// TwinCAT 3 PLC project HOMS_XRT_PLC
// Title: lcls-plc-xrt-optics
// Company: SLAC
// ProjectVersion: 5.7.0
// ProgramVersion: 3.1.4022.7
// CompilerDefines: L
// libraries:
//   lcls-twincat-motion, * (SLAC)
//   lcls-twincat-optics, * (SLAC)
//   PMPS, * (SLAC - LCLS)
//   Tc2_ControllerToolbox, * (Beckhoff Automation GmbH)
//   Tc2_EtherCAT, * (Beckhoff Automation GmbH)
//   Tc2_MC2, * (Beckhoff Automation GmbH)
//   Tc2_SerialCom, * (Beckhoff Automation GmbH)
//   Tc2_Standard, * (Beckhoff Automation GmbH)
//   Tc2_System, * (Beckhoff Automation GmbH)
//   Tc2_Utilities, * (Beckhoff Automation GmbH)
//   Tc3_Module, * (Beckhoff Automation GmbH)
//   VisuDialogs, * (System)
//   LCLS General,2.8.2,SLAC
// project tree:
//   Common/DUTs/ ENUM_Coating_States.TcDUT, E_GantryControl.TcDUT, E_GantryMode.TcDUT, E_PiezoControl.TcDUT, E_PitchControl.TcDUT, HOMS_Gantry.TcDUT, HOMS_GantryAxis.TcDUT, HOMS_PitchMechanismOld.TcDUT, ST_AbstractAxis.TcDUT, ST_CoEIndSub.TcDUT, ST_DecoupledMotionPermits.TcDUT, ST_ElmoGDCBellCoEParams.TcDUT, ST_HOMSStepper.TcDUT, ST_PiezoAxisOld.TcDUT, ST_StepperStatus.TcDUT
//   Version/ Global_Version.TcGVL
//   Common/POUs/Helpers/ FB_Drive.TcPOU, FB_ElmoGDCBellCoE.TcPOU, FB_ElmoMCUploadDriveParams.TcPOU, FB_ElmoStoMonitor.TcPOU, FB_GantryDiffVirtualLimitSwitch.TcPOU, FB_InitDriveRefs.TcPOU, FB_LimitSwitchState.TcPOU, FB_PitchSoftLimits.TcPOU, FB_PI_E621_SerialDriverOld.TcPOU, FB_PI_E621_SerialTransaction.TcPOU, FB_PTP.TcPOU, FB_ReadFloatParameter.TcPOU, FB_ReadParameterInNC.TcPOU, FB_WriteParameterInNC.TcPOU, F_PiezoPosition.TcPOU, MC_SmoothMover.TcPOU, WithinRange.TcPOU
//   Common/POUs/HOMS_FBs/ FB_Gantry.TcPOU, FB_GantryDifferenceMonitor.TcPOU, FB_PiezoControl.TcPOU, FB_PitchControlOld.TcPOU, FB_ReduceGantryDiff.TcPOU
//   / GlobalTextList.TcGTLO, PiezoDriver.TcTTO, PlcTask.TcTTO, SerialIO.TcTTO, Visualization Manager.TcVMO (not stored)
//   GVLs/ GVL.TcGVL, GVL_COM_Buffers.TcGVL, GVL_Constants.TcGVL, GVL_MR1L3.TcGVL, GVL_MR1L4_Constants.TcGVL, GVL_MR1L4.TcGVL, GVL_MR1L3_Constants.TcGVL, GVL_MR2L3_Constants.TcGVL, GVL_MR2L3.TcGVL, GVL_PMPS.TcGVL, GVL_RTDS.TcGVL, GVL_SerialIO.TcGVL
//   POUs/ FB_Coating_States_noPMPS.TcPOU, FB_MirrorCoatingProtection.TcPOU, FB_Coating_States.TcPOU, Main.TcPOU, PRG_PMPS.TcPOU, PRG_CoatingProtection.TcPOU, PRG_States.TcPOU
//   POUs/Serial Comm/ PiezoSerial.TcPOU, P_Serial_Com.TcPOU
//   VISUs/ GantryControls.TcVIS, Visualization.TcVIS, PiezoControls.TcVIS
// real-time tasks:
//   TASK PlcTask: cycle T#10ms, priority 20, ADS port 350
//   TASK SerialIO: cycle T#2ms, priority 1, ADS port 351
//   TASK LoggerTask: cycle T#10ms, priority 2, ADS port 352
//   TASK PiezoDriver: cycle T#1ms, priority 3, ADS port 353
// motion (NC):
//   TASK NC-Task 1 SAF: cycle T#2ms, priority 4, ADS port 501
//   TASK NC-Task 1 SVB: cycle T#10ms, priority 8, ADS port 511
//   AXIS M1L3-Yup (id 1)
//     General: UnitName=um
//     Dynamic: Acceleration=200, Deceleration=200, DelayTime=0.008
//     Velo: Maximum=200
//     OtherSettings: AllowMotionCmdToSlave=true
//     encoder EncType=29
//       EncPara: ScaleFactorNumerator=0.001, Offset=-13611, MaxCount=#xffffffff
//         SoftEndMinControl: Enable=true, Range=-12130
//         SoftEndMaxControl: Enable=true, Range=12932
//         Inc: RefSoftSyncMask=#x0000ffff
//     drive DrvType=24
//       DrvPara: Inverse=true
//         Analog: VeloReferenz=488.28125, ScaleFactorActTorque=0.1
//         TimeComp: TaskDelayCycles=1
//     controller CtrType=2
//       CtrPara: PriorControlFactor=1
//         PosDiffControl: Range=100
//         PID: PosKp=50, PosExtKp=10, DeadBandPosition=0.3
//         Observer: BandWidth=20
//   AXIS M1L3-Ydwn (id 2)
//     General: UnitName=um
//     Dynamic: Acceleration=200, Deceleration=200, DelayTime=0.008
//     Velo: Maximum=200
//     OtherSettings: AllowMotionCmdToSlave=true
//     encoder EncType=29
//       EncPara: ScaleFactorNumerator=0.001, Offset=-13433.6, MaxCount=#xffffffff
//         SoftEndMinControl: Enable=true, Range=-12130
//         SoftEndMaxControl: Enable=true, Range=12932
//         Inc: RefSoftSyncMask=#x0000ffff
//     drive DrvType=24
//       DrvPara: Inverse=true
//         Analog: VeloReferenz=488.28125, ScaleFactorActTorque=0.1
//         TimeComp: TaskDelayCycles=1
//     controller CtrType=2
//       CtrPara: PriorControlFactor=1
//         PosDiffControl: Range=100
//         PID: PosKp=50, PosExtKp=10, DeadBandPosition=0.3
//         Observer: BandWidth=20
//   AXIS M1L3-Xup (id 3)
//     General: UnitName=um
//     Dynamic: Acceleration=2000, Deceleration=2000, DelayTime=0.008
//     Velo: Maximum=1000
//     OtherSettings: AllowMotionCmdToSlave=true
//     encoder EncType=29
//       EncPara: ScaleFactorNumerator=0.001, Offset=-25210.5, MaxCount=#xffffffff
//         SoftEndMinControl: Enable=true, Range=-6841
//         SoftEndMaxControl: Enable=true, Range=1452.7
//         Inc: RefSoftSyncMask=#x0000ffff
//     drive DrvType=24
//       Analog: VeloReferenz=1220.703125, ScaleFactorActTorque=0.1
//       TimeComp: TaskDelayCycles=1
//     controller CtrType=2
//       CtrPara: PriorControlFactor=1
//         PosDiffControl: Range=50
//         PID: PosKp=50, PosExtKp=50, DeadBandPosition=0.4
//         Observer: BandWidth=20
//   AXIS M1L3-Xdwn (id 4)
//     General: UnitName=um
//     Dynamic: Acceleration=2000, Deceleration=2000, DelayTime=0.008
//     Velo: Maximum=1000
//     OtherSettings: AllowMotionCmdToSlave=true
//     encoder EncType=29
//       EncPara: ScaleFactorNumerator=0.001, Offset=-24971.8, MaxCount=#xffffffff
//         SoftEndMinControl: Enable=true, Range=-6841.9
//         SoftEndMaxControl: Enable=true, Range=1452.7
//         Inc: RefSoftSyncMask=#x0000ffff
//     drive DrvType=24
//       DrvPara: Inverse=true
//         Analog: VeloReferenz=1220.703125, ScaleFactorActTorque=0.1
//         TimeComp: TaskDelayCycles=1
//     controller CtrType=2
//       CtrPara: PriorControlFactor=1
//         PosDiffControl: Range=50
//         PID: PosKp=50, PosExtKp=50, DeadBandPosition=0.4
//         Observer: BandWidth=20
//   AXIS M1L3-Pitch (id 5)
//     General: UnitName=urad
//     Dynamic: Acceleration=390, Deceleration=390, DelayTime=0.008
//     Velo: Maximum=150
//     OtherSettings: AllowMotionCmdToSlave=true
//     encoder EncType=29
//       EncPara: ScaleFactorNumerator=0.001949317739, Offset=-21644.29, MaxCount=#xffffffff
//         FilterTime: TPos=0.2
//         SoftEndMinControl: Enable=true, Range=-193
//         SoftEndMaxControl: Enable=true, Range=220
//         Inc: RefSoftSyncMask=#x0000ffff
//     drive DrvType=24
//       Analog: VeloReferenz=371.8028524, ScaleFactorActTorque=0.1
//       TimeComp: TaskDelayCycles=1
//     controller CtrType=2
//       CtrPara: PriorControlFactor=1
//         PosDiffControl: Range=30
//         PID: PosKp=2, PosExtKp=1, DeadBandPosition=0.01
//         Observer: BandWidth=20
//   AXIS M1L3-Bender (id 6)
//     General: UnitName=um
//     Dynamic: Acceleration=150, Deceleration=150, DelayTime=0.008
//     Velo: Maximum=150
//     OtherSettings: AllowMotionCmdToSlave=true
//     encoder EncType=29
//       EncPara: ScaleFactorNumerator=0.001, MaxCount=#xffffffff
//         SoftEndMinControl: Enable=true, Range=18000
//         SoftEndMaxControl: Enable=true, Range=27800
//         Inc: RefSoftSyncMask=#x0000ffff
//     drive DrvType=24
//       DrvPara: Inverse=true
//         Analog: VeloReferenz=150, ScaleFactorActTorque=0.1
//         TimeComp: TaskDelayCycles=1
//     controller CtrType=2
//       CtrPara: PriorControlFactor=1
//         PID: PosKp=10, PosExtKp=0.001, PosExtVelo=0.9, DeadBandPosition=0.1
//         Observer: BandWidth=20
//   AXIS M2L3-Yup (id 13)
//     General: UnitName=um
//     Dynamic: Acceleration=200, Deceleration=200, DelayTime=0.008
//     Velo: Maximum=200
//     OtherSettings: AllowMotionCmdToSlave=true
//     encoder EncType=29
//       EncPara: ScaleFactorNumerator=0.001, Offset=-14279, MaxCount=#xffffffff
//         SoftEndMinControl: Enable=true, Range=-11750
//         SoftEndMaxControl: Enable=true, Range=12530
//         Inc: RefSoftSyncMask=#x0000ffff
//     drive DrvType=24
//       DrvPara: Inverse=true
//         Analog: VeloReferenz=488.28125, ScaleFactorActTorque=0.1
//         TimeComp: TaskDelayCycles=1
//     controller CtrType=2
//       CtrPara: PriorControlFactor=1
//         PosDiffControl: Range=100
//         PID: PosKp=50, PosExtKp=10, DeadBandPosition=0.3
//         Observer: BandWidth=20
//   AXIS M2L3-Ydwn (id 14)
//     General: UnitName=um
//     Dynamic: Acceleration=200, Deceleration=200, DelayTime=0.008
//     Velo: Maximum=200
//     OtherSettings: AllowMotionCmdToSlave=true
//     encoder EncType=29
//       EncPara: ScaleFactorNumerator=0.001, Offset=-16314.1, MaxCount=#xffffffff
//         SoftEndMinControl: Enable=true, Range=-11750
//         SoftEndMaxControl: Enable=true, Range=12531.5
//         Inc: RefSoftSyncMask=#x0000ffff
//     drive DrvType=24
//       DrvPara: Inverse=true
//         Analog: VeloReferenz=488.28125, ScaleFactorActTorque=0.1
//         TimeComp: TaskDelayCycles=1
//     controller CtrType=2
//       CtrPara: PriorControlFactor=1
//         PosDiffControl: Range=100
//         PID: PosKp=50, PosExtKp=10, DeadBandPosition=0.3
//         Observer: BandWidth=20
//   AXIS M2L3-Xup (id 15)
//     General: UnitName=um
//     Dynamic: Acceleration=2000, Deceleration=2000, DelayTime=0.008
//     Velo: Maximum=1000
//     OtherSettings: AllowMotionCmdToSlave=true
//     encoder EncType=29
//       EncPara: ScaleFactorNumerator=0.001, Offset=-25135.5, MaxCount=#xffffffff
//         SoftEndMinControl: Enable=true, Range=-850
//         SoftEndMaxControl: Enable=true, Range=867.4
//         Inc: RefSoftSyncMask=#x0000ffff
//     drive DrvType=24
//       Analog: VeloReferenz=1220.703125, ScaleFactorActTorque=0.1
//       TimeComp: TaskDelayCycles=1
//     controller CtrType=2
//       CtrPara: PriorControlFactor=1
//         PosDiffControl: Range=50
//         PID: PosKp=50, PosExtKp=50, DeadBandPosition=0.4
//         Observer: BandWidth=20
//   AXIS M2L3-Xdwn (id 16)
//     General: UnitName=um
//     Dynamic: Acceleration=2000, Deceleration=2000, DelayTime=0.008
//     Velo: Maximum=1000
//     OtherSettings: AllowMotionCmdToSlave=true
//     encoder EncType=29
//       EncPara: ScaleFactorNumerator=0.001, Offset=-24091, MaxCount=#xffffffff
//         SoftEndMinControl: Enable=true, Range=-865
//         SoftEndMaxControl: Enable=true, Range=862.6
//         Inc: RefSoftSyncMask=#x0000ffff
//     drive DrvType=24
//       DrvPara: Inverse=true
//         Analog: VeloReferenz=1220.703125, ScaleFactorActTorque=0.1
//         TimeComp: TaskDelayCycles=1
//     controller CtrType=2
//       CtrPara: PriorControlFactor=1
//         PosDiffControl: Range=50
//         PID: PosKp=50, PosExtKp=50, DeadBandPosition=0.4
//         Observer: BandWidth=20
//   AXIS M2L3-Pitch (id 17)
//     General: UnitName=urad
//     Dynamic: Acceleration=390, Deceleration=390, DelayTime=0.008
//     Velo: Maximum=150
//     OtherSettings: AllowMotionCmdToSlave=true
//     encoder EncType=29
//       EncPara: ScaleFactorNumerator=0.001949317739, Offset=-17539, MaxCount=#xffffffff
//         FilterTime: TPos=0.2
//         SoftEndMinControl: Enable=true, Range=-212
//         SoftEndMaxControl: Enable=true, Range=246
//         Inc: RefSoftSyncMask=#x0000ffff
//     drive DrvType=24
//       Analog: VeloReferenz=371.8028524, ScaleFactorActTorque=0.1
//       TimeComp: TaskDelayCycles=1
//     controller CtrType=2
//       CtrPara: PriorControlFactor=1
//         PosDiffControl: Range=15
//         PID: PosKp=2, PosExtKp=1, DeadBandPosition=0.01
//         Observer: BandWidth=20
//   AXIS M2L3-Bender (id 18)
//     General: UnitName=um
//     Dynamic: Acceleration=150, Deceleration=150, DelayTime=0.008
//     Velo: Maximum=150
//     OtherSettings: AllowMotionCmdToSlave=true
//     encoder EncType=29
//       EncPara: ScaleFactorNumerator=0.001, MaxCount=#xffffffff
//         SoftEndMinControl: Enable=true, Range=20000
//         SoftEndMaxControl: Enable=true, Range=32000
//         Inc: RefSoftSyncMask=#x0000ffff
//     drive DrvType=24
//       DrvPara: Inverse=true
//         Analog: VeloReferenz=195.3125, ScaleFactorActTorque=0.1
//         TimeComp: TaskDelayCycles=1
//     controller CtrType=2
//       CtrPara: PriorControlFactor=1
//         PID: PosKp=10, PosExtKp=0.001, PosExtVelo=0.9, DeadBandPosition=0.1
//         Observer: BandWidth=20
//   AXIS M1L4-Yup (id 7)
//     General: UnitName=um
//     Dynamic: Acceleration=200, Deceleration=200, DelayTime=0.008
//     Velo: Maximum=200
//     OtherSettings: AllowMotionCmdToSlave=true
//     encoder EncType=29
//       EncPara: ScaleFactorNumerator=0.001, Offset=-13496.029, MaxCount=#xffffffff
//         SoftEndMinControl: Enable=true, Range=-11000
//         SoftEndMaxControl: Enable=true, Range=12000
//         Inc: RefSoftSyncMask=#x0000ffff
//     drive DrvType=24
//       DrvPara: Inverse=true
//         Analog: VeloReferenz=488.28125, ScaleFactorActTorque=0.1
//         TimeComp: TaskDelayCycles=1
//     controller CtrType=2
//       CtrPara: PriorControlFactor=1
//         PosDiffControl: Range=100
//         PID: PosKp=50, PosExtKp=10, DeadBandPosition=0.3
//         Observer: BandWidth=20
//   AXIS M1L4-Ydwn (id 8)
//     General: UnitName=um
//     Dynamic: Acceleration=200, Deceleration=200, DelayTime=0.008
//     Velo: Maximum=200
//     OtherSettings: AllowMotionCmdToSlave=true
//     encoder EncType=29
//       EncPara: ScaleFactorNumerator=0.001, Offset=-14872.55, MaxCount=#xffffffff
//         SoftEndMinControl: Enable=true, Range=-11000
//         SoftEndMaxControl: Enable=true, Range=12075
//         Inc: RefSoftSyncMask=#x0000ffff
//     drive DrvType=24
//       DrvPara: Inverse=true
//         Analog: VeloReferenz=488.28125, ScaleFactorActTorque=0.1
//         TimeComp: TaskDelayCycles=1
//     controller CtrType=2
//       CtrPara: PriorControlFactor=1
//         PosDiffControl: Range=100
//         PID: PosKp=50, PosExtKp=10, DeadBandPosition=0.3
//         Observer: BandWidth=20
//   AXIS M1L4-Xup (id 9)
//     General: UnitName=um
//     Dynamic: Acceleration=2000, Deceleration=2000, DelayTime=0.008
//     Velo: Maximum=1000
//     OtherSettings: AllowMotionCmdToSlave=true
//     encoder EncType=29
//       EncPara: ScaleFactorNumerator=0.001, Offset=-25490.849, MaxCount=#xffffffff
//         SoftEndMinControl: Enable=true, Range=-2000
//         SoftEndMaxControl: Enable=true, Range=18750
//         Inc: RefSoftSyncMask=#x0000ffff
//     drive DrvType=24
//       Analog: VeloReferenz=1220.703125, ScaleFactorActTorque=0.1
//       TimeComp: TaskDelayCycles=1
//     controller CtrType=2
//       CtrPara: PriorControlFactor=1
//         PosDiffControl: Range=50
//         PID: PosKp=50, PosExtKp=50, DeadBandPosition=0.4
//         Observer: BandWidth=20
//   AXIS M1L4-Xdwn (id 10)
//     General: UnitName=um
//     Dynamic: Acceleration=2000, Deceleration=2000, DelayTime=0.008
//     Velo: Maximum=1000
//     OtherSettings: AllowMotionCmdToSlave=true
//     encoder EncType=29
//       EncPara: ScaleFactorNumerator=0.001, Offset=-26628.83, MaxCount=#xffffffff
//         SoftEndMinControl: Enable=true, Range=-2050
//         SoftEndMaxControl: Enable=true, Range=18750
//         Inc: RefSoftSyncMask=#x0000ffff
//     drive DrvType=24
//       DrvPara: Inverse=true
//         Analog: VeloReferenz=1220.703125, ScaleFactorActTorque=0.1
//         TimeComp: TaskDelayCycles=1
//     controller CtrType=2
//       CtrPara: PriorControlFactor=1
//         PosDiffControl: Range=50
//         PID: PosKp=50, PosExtKp=50, DeadBandPosition=0.4
//         Observer: BandWidth=20
//   AXIS M1L4-Pitch (id 11)
//     General: UnitName=urad
//     Dynamic: Acceleration=390, Deceleration=390, DelayTime=0.008
//     Velo: Maximum=150
//     OtherSettings: AllowMotionCmdToSlave=true
//     encoder EncType=29
//       EncPara: ScaleFactorNumerator=0.001949317739, Offset=-19152.5, MaxCount=#xffffffff
//         FilterTime: TPos=0.2
//         SoftEndMinControl: Enable=true, Range=-900
//         SoftEndMaxControl: Enable=true, Range=900
//         Inc: RefSoftSyncMask=#x0000ffff
//     drive DrvType=24
//       Analog: VeloReferenz=371.8028524, ScaleFactorActTorque=0.1
//       TimeComp: TaskDelayCycles=1
//     controller CtrType=2
//       CtrPara: PriorControlFactor=1
//         PosDiffControl: Range=30
//         PID: PosKp=2, PosExtKp=1, DeadBandPosition=0.01
//         Observer: BandWidth=20
//   AXIS M1L4-Bender (id 12)
//     General: UnitName=um
//     Dynamic: AccelerationMaximum=50, DecelerationMaximum=50, Acceleration=50, Deceleration=50, DelayTime=0.008
//     Velo: Maximum=150
//     OtherSettings: AllowMotionCmdToSlave=true
//     encoder EncType=29
//       EncPara: ScaleFactorNumerator=0.001, Offset=-4295012.99, MaxCount=#xffffffff
//         SoftEndMinControl: Enable=true, Range=-26500
//         SoftEndMaxControl: Enable=true, Range=-16500
//     drive DrvType=24
//       DrvPara: Inverse=true
//         Analog: VeloReferenz=195.3125, ScaleFactorActTorque=0.1
//         TimeComp: TaskDelayCycles=1
//     controller CtrType=2
//       CtrPara: PriorControlFactor=1
//         PosDiffControl: Range=100
//         PID: PosKp=10, PosExtKp=0.001, PosExtVelo=0.9, DeadBandPosition=0.1
//         Observer: BandWidth=20
// I/O:
//   DEVICE HOMS, AmsNetId 172.21.88.136.2.1
//     Term 1 (EK1200) [EK1200-5000 EtherCAT Power supply (2A E-Bus)]
//       Term 24 (EL9187) [EL9187 Potential Connection, 8 x Ground]
//       Term 13 (EL2008) [EL2008 8Ch. Dig. Output 24V, 0.5A]
//       Term 14 (EK1122) [EK1122 2 port EtherCAT junction]
//         EK1100_M1L3 [EK1100 EtherCAT Coupler (2A E-Bus)]
//           EL7041-1000_M1L3_Xup [EL7041-1000 1Ch. Stepper motor output stage (50V, 5A, standard)]
//           EL7041-1000_M1L3_Xdwn [EL7041-1000 1Ch. Stepper motor output stage (50V, 5A, standard)]
//           EL7041-1000_M1L3_Yup [EL7041-1000 1Ch. Stepper motor output stage (50V, 5A, standard)]
//           EL7041-1000_M1L3_Ydwn [EL7041-1000 1Ch. Stepper motor output stage (50V, 5A, standard)]
//           EL7041-1000_M1L3_PitchCoarse [EL7041-1000 1Ch. Stepper motor output stage (50V, 5A, standard)]
//           EL7041-1000_M1L3_Bender
//           EL6001_M1L3_PitchFine [EL6001 Interface (RS232)]
//           EL5042_M1L3_Xupdwn
//           EL5042_M1L3_Yupdwn
//           EL5042_M1L3_PitchBender
//           EL1004_M1L3_STO
//           EL9505_M1L3_BenderLims
//           MR1L3-EL3202-0010-E13
//           MR1L3-EL3202-0010-E14
//           Term 42 (EL9011)
//         EK1100_M1L4 [EK1100 EtherCAT Coupler (2A E-Bus)]
//           EL7041-1000_M1L4_Xup [EL7041-1000 1Ch. Stepper motor output stage (50V, 5A, standard)]
//           EL7041-1000_M1L4_Xdwn [EL7041-1000 1Ch. Stepper motor output stage (50V, 5A, standard)]
//           EL7041-1000_M1L4_Yup [EL7041-1000 1Ch. Stepper motor output stage (50V, 5A, standard)]
//           EL7041-1000_M1L4_Ydwn [EL7041-1000 1Ch. Stepper motor output stage (50V, 5A, standard)]
//           EL7041-1000_M1L4_PitchCoarse [EL7041-1000 1Ch. Stepper motor output stage (50V, 5A, standard)]
//           EL7041-1000_M1L4_Bender
//           EL6001_M1L4_PitchFine [EL6001 Interface (RS232)]
//           EL5042_M1L4_Xupdwn
//           EL5042_M1L4_Yupdwn
//           EL5042_M1L4_PitchBender
//           EL1004_M1L4_STO
//           EL9505_M1L4_BenderLims
//           MR1L4-EL3202-0010-E13
//           MR1L4-EL3202-0010-E14
//           Term 29 (EL9011)
//       Term 2 (EK1122) [EK1122 2 port EtherCAT junction]
//         EK1100_M2L3
//       Term 34 (EK1521-0010)
// variable links:
//   (this object) <-> HOMS/Term 1 (EK1200)/Term 14 (EK1122)/EK1100_M1L3/EL5042_M1L3_Yupdwn
//     Enc/Inputs/In/nComState @bit 1 <-> WcState/InputToggle
//     Enc/Inputs/In/nComState <-> WcState/WcState
//     Enc/Inputs/In/nDataIn1 <-> FB Inputs Channel 1/Position
//     Enc/Inputs/In/nDataIn1 <-> FB Inputs Channel 2/Position
//     Enc/Inputs/In/nState1 @bit 12 <-> FB Inputs Channel 1/Status/Diag
//     Enc/Inputs/In/nState1 @bit 12 <-> FB Inputs Channel 2/Status/Diag
//     Enc/Inputs/In/nState1 @bit 1 <-> FB Inputs Channel 1/Status/Error
//     Enc/Inputs/In/nState1 @bit 1 <-> FB Inputs Channel 2/Status/Error
//     Enc/Inputs/In/nState1 @bit 14 <-> FB Inputs Channel 1/Status/Input cycle counter
//     Enc/Inputs/In/nState1 @bit 14 <-> FB Inputs Channel 2/Status/Input cycle counter
//     Enc/Inputs/In/nState1 @bit 2 <-> FB Inputs Channel 1/Status/Ready
//     Enc/Inputs/In/nState1 @bit 2 <-> FB Inputs Channel 2/Status/Ready
//     Enc/Inputs/In/nState1 @bit 13 <-> FB Inputs Channel 1/Status/TxPDO State
//     Enc/Inputs/In/nState1 @bit 13 <-> FB Inputs Channel 2/Status/TxPDO State
//     Enc/Inputs/In/nState1 <-> FB Inputs Channel 1/Status/Warning
//     Enc/Inputs/In/nState1 <-> FB Inputs Channel 2/Status/Warning
//   (this object) <-> HOMS/Term 1 (EK1200)/Term 14 (EK1122)/EK1100_M1L3/EL7041-1000_M1L3_Yup
//     Drive/Inputs/In/nState1 @bit 3 <-> STM Status/Status/Error
//     Drive/Inputs/In/nState1 @bit 5 <-> STM Status/Status/Moving negative
//     Drive/Inputs/In/nState1 @bit 4 <-> STM Status/Status/Moving positive
//     Drive/Inputs/In/nState1 @bit 1 <-> STM Status/Status/Ready
//     Drive/Inputs/In/nState1 <-> STM Status/Status/Ready to enable
//     Drive/Inputs/In/nState1 @bit 6 <-> STM Status/Status/Torque reduced
//     Drive/Inputs/In/nState1 @bit 2 <-> STM Status/Status/Warning
//     Drive/Inputs/In/nState2 @bit 3 <-> STM Status/Status/Digital input 1
//     Drive/Inputs/In/nState2 @bit 4 <-> STM Status/Status/Digital input 2
//     Drive/Inputs/In/nState2 @bit 5 <-> STM Status/Status/Sync error
//     Drive/Inputs/In/nState2 @bit 7 <-> STM Status/Status/TxPDO Toggle
//     Drive/Inputs/In/nState4 @bit 1 <-> WcState/InputToggle
//     Drive/Inputs/In/nState4 <-> WcState/WcState
//     Drive/Outputs/Out/nCtrl1 <-> STM Control/Control/Enable
//     Drive/Outputs/Out/nCtrl1 @bit 2 <-> STM Control/Control/Reduce torque
//     Drive/Outputs/Out/nCtrl1 @bit 1 <-> STM Control/Control/Reset
//     Drive/Outputs/Out/nDataOut2[0] <-> STM Velocity/Velocity
//   (this object) <-> HOMS/Term 1 (EK1200)/Term 14 (EK1122)/EK1100_M1L3/EL7041-1000_M1L3_Ydwn
//     Drive/Inputs/In/nState1 @bit 3 <-> STM Status/Status/Error
//     Drive/Inputs/In/nState1 @bit 5 <-> STM Status/Status/Moving negative
//     Drive/Inputs/In/nState1 @bit 4 <-> STM Status/Status/Moving positive
//     Drive/Inputs/In/nState1 @bit 1 <-> STM Status/Status/Ready
//     Drive/Inputs/In/nState1 <-> STM Status/Status/Ready to enable
//     Drive/Inputs/In/nState1 @bit 6 <-> STM Status/Status/Torque reduced
//     Drive/Inputs/In/nState1 @bit 2 <-> STM Status/Status/Warning
//     Drive/Inputs/In/nState2 @bit 3 <-> STM Status/Status/Digital input 1
//     Drive/Inputs/In/nState2 @bit 4 <-> STM Status/Status/Digital input 2
//     Drive/Inputs/In/nState2 @bit 5 <-> STM Status/Status/Sync error
//     Drive/Inputs/In/nState2 @bit 7 <-> STM Status/Status/TxPDO Toggle
//     Drive/Inputs/In/nState4 @bit 1 <-> WcState/InputToggle
//     Drive/Inputs/In/nState4 <-> WcState/WcState
//     Drive/Outputs/Out/nCtrl1 <-> STM Control/Control/Enable
//     Drive/Outputs/Out/nCtrl1 @bit 2 <-> STM Control/Control/Reduce torque
//     Drive/Outputs/Out/nCtrl1 @bit 1 <-> STM Control/Control/Reset
//     Drive/Outputs/Out/nDataOut2[0] <-> STM Velocity/Velocity
//   (this object) <-> HOMS/Term 1 (EK1200)/Term 14 (EK1122)/EK1100_M1L3/EL5042_M1L3_Xupdwn
//     Enc/Inputs/In/nComState @bit 1 <-> WcState/InputToggle
//     Enc/Inputs/In/nComState <-> WcState/WcState
//     Enc/Inputs/In/nDataIn1 <-> FB Inputs Channel 1/Position
//     Enc/Inputs/In/nDataIn1 <-> FB Inputs Channel 2/Position
//     Enc/Inputs/In/nState1 @bit 12 <-> FB Inputs Channel 1/Status/Diag
//     Enc/Inputs/In/nState1 @bit 12 <-> FB Inputs Channel 2/Status/Diag
//     Enc/Inputs/In/nState1 @bit 1 <-> FB Inputs Channel 1/Status/Error
//     Enc/Inputs/In/nState1 @bit 1 <-> FB Inputs Channel 2/Status/Error
//     Enc/Inputs/In/nState1 @bit 14 <-> FB Inputs Channel 1/Status/Input cycle counter
//     Enc/Inputs/In/nState1 @bit 14 <-> FB Inputs Channel 2/Status/Input cycle counter
//     Enc/Inputs/In/nState1 @bit 2 <-> FB Inputs Channel 1/Status/Ready
//     Enc/Inputs/In/nState1 @bit 2 <-> FB Inputs Channel 2/Status/Ready
//     Enc/Inputs/In/nState1 @bit 13 <-> FB Inputs Channel 1/Status/TxPDO State
//     Enc/Inputs/In/nState1 @bit 13 <-> FB Inputs Channel 2/Status/TxPDO State
//     Enc/Inputs/In/nState1 <-> FB Inputs Channel 1/Status/Warning
//     Enc/Inputs/In/nState1 <-> FB Inputs Channel 2/Status/Warning
//   (this object) <-> HOMS/Term 1 (EK1200)/Term 14 (EK1122)/EK1100_M1L3/EL7041-1000_M1L3_Xup
//     Drive/Inputs/In/nState1 @bit 3 <-> STM Status/Status/Error
//     Drive/Inputs/In/nState1 @bit 5 <-> STM Status/Status/Moving negative
//     Drive/Inputs/In/nState1 @bit 4 <-> STM Status/Status/Moving positive
//     Drive/Inputs/In/nState1 @bit 1 <-> STM Status/Status/Ready
//     Drive/Inputs/In/nState1 <-> STM Status/Status/Ready to enable
//     Drive/Inputs/In/nState1 @bit 6 <-> STM Status/Status/Torque reduced
//     Drive/Inputs/In/nState1 @bit 2 <-> STM Status/Status/Warning
//     Drive/Inputs/In/nState2 @bit 3 <-> STM Status/Status/Digital input 1
//     Drive/Inputs/In/nState2 @bit 4 <-> STM Status/Status/Digital input 2
//     Drive/Inputs/In/nState2 @bit 5 <-> STM Status/Status/Sync error
//     Drive/Inputs/In/nState2 @bit 7 <-> STM Status/Status/TxPDO Toggle
//     Drive/Inputs/In/nState4 @bit 1 <-> WcState/InputToggle
//     Drive/Inputs/In/nState4 <-> WcState/WcState
//     Drive/Outputs/Out/nCtrl1 <-> STM Control/Control/Enable
//     Drive/Outputs/Out/nCtrl1 @bit 2 <-> STM Control/Control/Reduce torque
//     Drive/Outputs/Out/nCtrl1 @bit 1 <-> STM Control/Control/Reset
//     Drive/Outputs/Out/nDataOut2[0] <-> STM Velocity/Velocity
//   (this object) <-> HOMS/Term 1 (EK1200)/Term 14 (EK1122)/EK1100_M1L3/EL7041-1000_M1L3_Xdwn
//     Drive/Inputs/In/nState1 @bit 3 <-> STM Status/Status/Error
//     Drive/Inputs/In/nState1 @bit 5 <-> STM Status/Status/Moving negative
//     Drive/Inputs/In/nState1 @bit 4 <-> STM Status/Status/Moving positive
//     Drive/Inputs/In/nState1 @bit 1 <-> STM Status/Status/Ready
//     Drive/Inputs/In/nState1 <-> STM Status/Status/Ready to enable
//     Drive/Inputs/In/nState1 @bit 6 <-> STM Status/Status/Torque reduced
//     Drive/Inputs/In/nState1 @bit 2 <-> STM Status/Status/Warning
//     Drive/Inputs/In/nState2 @bit 3 <-> STM Status/Status/Digital input 1
//     Drive/Inputs/In/nState2 @bit 4 <-> STM Status/Status/Digital input 2
//     Drive/Inputs/In/nState2 @bit 5 <-> STM Status/Status/Sync error
//     Drive/Inputs/In/nState2 @bit 7 <-> STM Status/Status/TxPDO Toggle
//     Drive/Inputs/In/nState4 @bit 1 <-> WcState/InputToggle
//     Drive/Inputs/In/nState4 <-> WcState/WcState
//     Drive/Outputs/Out/nCtrl1 <-> STM Control/Control/Enable
//     Drive/Outputs/Out/nCtrl1 @bit 2 <-> STM Control/Control/Reduce torque
//     Drive/Outputs/Out/nCtrl1 @bit 1 <-> STM Control/Control/Reset
//     Drive/Outputs/Out/nDataOut2[0] <-> STM Velocity/Velocity
//   (this object) <-> HOMS/Term 1 (EK1200)/Term 14 (EK1122)/EK1100_M1L3/EL5042_M1L3_PitchBender
//     Enc/Inputs/In/nComState @bit 1 <-> WcState/InputToggle
//     Enc/Inputs/In/nComState <-> WcState/WcState
//     Enc/Inputs/In/nDataIn1 <-> FB Inputs Channel 1/Position
//     Enc/Inputs/In/nDataIn1 <-> FB Inputs Channel 2/Position
//     Enc/Inputs/In/nState1 @bit 12 <-> FB Inputs Channel 1/Status/Diag
//     Enc/Inputs/In/nState1 @bit 12 <-> FB Inputs Channel 2/Status/Diag
//     Enc/Inputs/In/nState1 @bit 1 <-> FB Inputs Channel 1/Status/Error
//     Enc/Inputs/In/nState1 @bit 1 <-> FB Inputs Channel 2/Status/Error
//     Enc/Inputs/In/nState1 @bit 14 <-> FB Inputs Channel 1/Status/Input cycle counter
//     Enc/Inputs/In/nState1 @bit 14 <-> FB Inputs Channel 2/Status/Input cycle counter
//     Enc/Inputs/In/nState1 @bit 2 <-> FB Inputs Channel 1/Status/Ready
//     Enc/Inputs/In/nState1 @bit 2 <-> FB Inputs Channel 2/Status/Ready
//     Enc/Inputs/In/nState1 @bit 13 <-> FB Inputs Channel 1/Status/TxPDO State
//     Enc/Inputs/In/nState1 @bit 13 <-> FB Inputs Channel 2/Status/TxPDO State
//     Enc/Inputs/In/nState1 <-> FB Inputs Channel 1/Status/Warning
//     Enc/Inputs/In/nState1 <-> FB Inputs Channel 2/Status/Warning
//   (this object) <-> HOMS/Term 1 (EK1200)/Term 14 (EK1122)/EK1100_M1L3/EL7041-1000_M1L3_PitchCoarse
//     Drive/Inputs/In/nState1 @bit 3 <-> STM Status/Status/Error
//     Drive/Inputs/In/nState1 @bit 5 <-> STM Status/Status/Moving negative
//     Drive/Inputs/In/nState1 @bit 4 <-> STM Status/Status/Moving positive
//     Drive/Inputs/In/nState1 @bit 1 <-> STM Status/Status/Ready
//     Drive/Inputs/In/nState1 <-> STM Status/Status/Ready to enable
//     Drive/Inputs/In/nState1 @bit 6 <-> STM Status/Status/Torque reduced
//     Drive/Inputs/In/nState1 @bit 2 <-> STM Status/Status/Warning
//     Drive/Inputs/In/nState2 @bit 3 <-> STM Status/Status/Digital input 1
//     Drive/Inputs/In/nState2 @bit 4 <-> STM Status/Status/Digital input 2
//     Drive/Inputs/In/nState2 @bit 5 <-> STM Status/Status/Sync error
//     Drive/Inputs/In/nState2 @bit 7 <-> STM Status/Status/TxPDO Toggle
//     Drive/Inputs/In/nState4 @bit 1 <-> WcState/InputToggle
//     Drive/Inputs/In/nState4 <-> WcState/WcState
//     Drive/Outputs/Out/nCtrl1 <-> STM Control/Control/Enable
//     Drive/Outputs/Out/nCtrl1 @bit 2 <-> STM Control/Control/Reduce torque
//     Drive/Outputs/Out/nCtrl1 @bit 1 <-> STM Control/Control/Reset
//     Drive/Outputs/Out/nDataOut2[0] <-> STM Velocity/Velocity
//   (this object) <-> HOMS/Term 1 (EK1200)/Term 14 (EK1122)/EK1100_M1L3/EL7041-1000_M1L3_Bender
//     Drive/Inputs/In/nState1 @bit 3 <-> STM Status/Status/Error
//     Drive/Inputs/In/nState1 @bit 5 <-> STM Status/Status/Moving negative
//     Drive/Inputs/In/nState1 @bit 4 <-> STM Status/Status/Moving positive
//     Drive/Inputs/In/nState1 @bit 1 <-> STM Status/Status/Ready
//     Drive/Inputs/In/nState1 <-> STM Status/Status/Ready to enable
//     Drive/Inputs/In/nState1 @bit 6 <-> STM Status/Status/Torque reduced
//     Drive/Inputs/In/nState1 @bit 2 <-> STM Status/Status/Warning
//     Drive/Inputs/In/nState2 @bit 3 <-> STM Status/Status/Digital input 1
//     Drive/Inputs/In/nState2 @bit 4 <-> STM Status/Status/Digital input 2
//     Drive/Inputs/In/nState2 @bit 5 <-> STM Status/Status/Sync error
//     Drive/Inputs/In/nState2 @bit 7 <-> STM Status/Status/TxPDO Toggle
//     Drive/Inputs/In/nState4 @bit 1 <-> WcState/InputToggle
//     Drive/Inputs/In/nState4 <-> WcState/WcState
//     Drive/Outputs/Out/nCtrl1 <-> STM Control/Control/Enable
//     Drive/Outputs/Out/nCtrl1 @bit 2 <-> STM Control/Control/Reduce torque
//     Drive/Outputs/Out/nCtrl1 @bit 1 <-> STM Control/Control/Reset
//     Drive/Outputs/Out/nDataOut2[0] <-> STM Velocity/Velocity
//   (this object) <-> HOMS/Term 1 (EK1200)/Term 2 (EK1122)/EK1100_M2L3/EL5042_M2L3_Yupdwn
//     Enc/Inputs/In/nComState @bit 1 <-> WcState/InputToggle
//     Enc/Inputs/In/nComState <-> WcState/WcState
//     Enc/Inputs/In/nDataIn1 <-> FB Inputs Channel 1/Position
//     Enc/Inputs/In/nDataIn1 <-> FB Inputs Channel 2/Position
//     Enc/Inputs/In/nState1 @bit 12 <-> FB Inputs Channel 1/Status/Diag
//     Enc/Inputs/In/nState1 @bit 12 <-> FB Inputs Channel 2/Status/Diag
//     Enc/Inputs/In/nState1 @bit 1 <-> FB Inputs Channel 1/Status/Error
//     Enc/Inputs/In/nState1 @bit 1 <-> FB Inputs Channel 2/Status/Error
//     Enc/Inputs/In/nState1 @bit 14 <-> FB Inputs Channel 1/Status/Input cycle counter
//     Enc/Inputs/In/nState1 @bit 14 <-> FB Inputs Channel 2/Status/Input cycle counter
//     Enc/Inputs/In/nState1 @bit 2 <-> FB Inputs Channel 1/Status/Ready
//     Enc/Inputs/In/nState1 @bit 2 <-> FB Inputs Channel 2/Status/Ready
//     Enc/Inputs/In/nState1 @bit 13 <-> FB Inputs Channel 1/Status/TxPDO State
//     Enc/Inputs/In/nState1 @bit 13 <-> FB Inputs Channel 2/Status/TxPDO State
//     Enc/Inputs/In/nState1 <-> FB Inputs Channel 1/Status/Warning
//     Enc/Inputs/In/nState1 <-> FB Inputs Channel 2/Status/Warning
//   (this object) <-> HOMS/Term 1 (EK1200)/Term 2 (EK1122)/EK1100_M2L3/EL7041-1000_M2L3_Yup
//     Drive/Inputs/In/nState1 @bit 3 <-> STM Status/Status/Error
//     Drive/Inputs/In/nState1 @bit 5 <-> STM Status/Status/Moving negative
//     Drive/Inputs/In/nState1 @bit 4 <-> STM Status/Status/Moving positive
//     Drive/Inputs/In/nState1 @bit 1 <-> STM Status/Status/Ready
//     Drive/Inputs/In/nState1 <-> STM Status/Status/Ready to enable
//     Drive/Inputs/In/nState1 @bit 6 <-> STM Status/Status/Torque reduced
//     Drive/Inputs/In/nState1 @bit 2 <-> STM Status/Status/Warning
//     Drive/Inputs/In/nState2 @bit 3 <-> STM Status/Status/Digital input 1
//     Drive/Inputs/In/nState2 @bit 4 <-> STM Status/Status/Digital input 2
//     Drive/Inputs/In/nState2 @bit 5 <-> STM Status/Status/Sync error
//     Drive/Inputs/In/nState2 @bit 7 <-> STM Status/Status/TxPDO Toggle
//     Drive/Inputs/In/nState4 @bit 1 <-> WcState/InputToggle
//     Drive/Inputs/In/nState4 <-> WcState/WcState
//     Drive/Outputs/Out/nCtrl1 <-> STM Control/Control/Enable
//     Drive/Outputs/Out/nCtrl1 @bit 2 <-> STM Control/Control/Reduce torque
//     Drive/Outputs/Out/nCtrl1 @bit 1 <-> STM Control/Control/Reset
//     Drive/Outputs/Out/nDataOut2[0] <-> STM Velocity/Velocity
//   (this object) <-> HOMS/Term 1 (EK1200)/Term 2 (EK1122)/EK1100_M2L3/EL7041-1000_M2L3_Ydwn
//     Drive/Inputs/In/nState1 @bit 3 <-> STM Status/Status/Error
//     Drive/Inputs/In/nState1 @bit 5 <-> STM Status/Status/Moving negative
//     Drive/Inputs/In/nState1 @bit 4 <-> STM Status/Status/Moving positive
//     Drive/Inputs/In/nState1 @bit 1 <-> STM Status/Status/Ready
//     Drive/Inputs/In/nState1 <-> STM Status/Status/Ready to enable
//     Drive/Inputs/In/nState1 @bit 6 <-> STM Status/Status/Torque reduced
//     Drive/Inputs/In/nState1 @bit 2 <-> STM Status/Status/Warning
//     Drive/Inputs/In/nState2 @bit 3 <-> STM Status/Status/Digital input 1
//     Drive/Inputs/In/nState2 @bit 4 <-> STM Status/Status/Digital input 2
//     Drive/Inputs/In/nState2 @bit 5 <-> STM Status/Status/Sync error
//     Drive/Inputs/In/nState2 @bit 7 <-> STM Status/Status/TxPDO Toggle
//     Drive/Inputs/In/nState4 @bit 1 <-> WcState/InputToggle
//     Drive/Inputs/In/nState4 <-> WcState/WcState
//     Drive/Outputs/Out/nCtrl1 <-> STM Control/Control/Enable
//     Drive/Outputs/Out/nCtrl1 @bit 2 <-> STM Control/Control/Reduce torque
//     Drive/Outputs/Out/nCtrl1 @bit 1 <-> STM Control/Control/Reset
//     Drive/Outputs/Out/nDataOut2[0] <-> STM Velocity/Velocity
//   (this object) <-> HOMS/Term 1 (EK1200)/Term 2 (EK1122)/EK1100_M2L3/EL5042_M2L3_Xupdwn
//     Enc/Inputs/In/nComState @bit 1 <-> WcState/InputToggle
//     Enc/Inputs/In/nComState <-> WcState/WcState
//     Enc/Inputs/In/nDataIn1 <-> FB Inputs Channel 1/Position
//     Enc/Inputs/In/nDataIn1 <-> FB Inputs Channel 2/Position
//     Enc/Inputs/In/nState1 @bit 12 <-> FB Inputs Channel 1/Status/Diag
//     Enc/Inputs/In/nState1 @bit 12 <-> FB Inputs Channel 2/Status/Diag
//     Enc/Inputs/In/nState1 @bit 1 <-> FB Inputs Channel 1/Status/Error
//     Enc/Inputs/In/nState1 @bit 1 <-> FB Inputs Channel 2/Status/Error
//     Enc/Inputs/In/nState1 @bit 14 <-> FB Inputs Channel 1/Status/Input cycle counter
//     Enc/Inputs/In/nState1 @bit 14 <-> FB Inputs Channel 2/Status/Input cycle counter
//     Enc/Inputs/In/nState1 @bit 2 <-> FB Inputs Channel 1/Status/Ready
//     Enc/Inputs/In/nState1 @bit 2 <-> FB Inputs Channel 2/Status/Ready
//     Enc/Inputs/In/nState1 @bit 13 <-> FB Inputs Channel 1/Status/TxPDO State
//     Enc/Inputs/In/nState1 @bit 13 <-> FB Inputs Channel 2/Status/TxPDO State
//     Enc/Inputs/In/nState1 <-> FB Inputs Channel 1/Status/Warning
//     Enc/Inputs/In/nState1 <-> FB Inputs Channel 2/Status/Warning
//   (this object) <-> HOMS/Term 1 (EK1200)/Term 2 (EK1122)/EK1100_M2L3/EL7041-1000_M2L3_Xup
//     Drive/Inputs/In/nState1 @bit 3 <-> STM Status/Status/Error
//     Drive/Inputs/In/nState1 @bit 5 <-> STM Status/Status/Moving negative
//     Drive/Inputs/In/nState1 @bit 4 <-> STM Status/Status/Moving positive
//     Drive/Inputs/In/nState1 @bit 1 <-> STM Status/Status/Ready
//     Drive/Inputs/In/nState1 <-> STM Status/Status/Ready to enable
//     Drive/Inputs/In/nState1 @bit 6 <-> STM Status/Status/Torque reduced
//     Drive/Inputs/In/nState1 @bit 2 <-> STM Status/Status/Warning
//     Drive/Inputs/In/nState2 @bit 3 <-> STM Status/Status/Digital input 1
//     Drive/Inputs/In/nState2 @bit 4 <-> STM Status/Status/Digital input 2
//     Drive/Inputs/In/nState2 @bit 5 <-> STM Status/Status/Sync error
//     Drive/Inputs/In/nState2 @bit 7 <-> STM Status/Status/TxPDO Toggle
//     Drive/Inputs/In/nState4 @bit 1 <-> WcState/InputToggle
//     Drive/Inputs/In/nState4 <-> WcState/WcState
//     Drive/Outputs/Out/nCtrl1 <-> STM Control/Control/Enable
//     Drive/Outputs/Out/nCtrl1 @bit 2 <-> STM Control/Control/Reduce torque
//     Drive/Outputs/Out/nCtrl1 @bit 1 <-> STM Control/Control/Reset
//     Drive/Outputs/Out/nDataOut2[0] <-> STM Velocity/Velocity
//   (this object) <-> HOMS/Term 1 (EK1200)/Term 2 (EK1122)/EK1100_M2L3/EL7041-1000_M2L3_Xdwn
//     Drive/Inputs/In/nState1 @bit 3 <-> STM Status/Status/Error
//     Drive/Inputs/In/nState1 @bit 5 <-> STM Status/Status/Moving negative
//     Drive/Inputs/In/nState1 @bit 4 <-> STM Status/Status/Moving positive
//     Drive/Inputs/In/nState1 @bit 1 <-> STM Status/Status/Ready
//     Drive/Inputs/In/nState1 <-> STM Status/Status/Ready to enable
//     Drive/Inputs/In/nState1 @bit 6 <-> STM Status/Status/Torque reduced
//     Drive/Inputs/In/nState1 @bit 2 <-> STM Status/Status/Warning
//     Drive/Inputs/In/nState2 @bit 3 <-> STM Status/Status/Digital input 1
//     Drive/Inputs/In/nState2 @bit 4 <-> STM Status/Status/Digital input 2
//     Drive/Inputs/In/nState2 @bit 5 <-> STM Status/Status/Sync error
//     Drive/Inputs/In/nState2 @bit 7 <-> STM Status/Status/TxPDO Toggle
//     Drive/Inputs/In/nState4 @bit 1 <-> WcState/InputToggle
//     Drive/Inputs/In/nState4 <-> WcState/WcState
//     Drive/Outputs/Out/nCtrl1 <-> STM Control/Control/Enable
//     Drive/Outputs/Out/nCtrl1 @bit 2 <-> STM Control/Control/Reduce torque
//     Drive/Outputs/Out/nCtrl1 @bit 1 <-> STM Control/Control/Reset
//     Drive/Outputs/Out/nDataOut2[0] <-> STM Velocity/Velocity
//   (this object) <-> HOMS/Term 1 (EK1200)/Term 2 (EK1122)/EK1100_M2L3/EL5042_M2L3_PitchBender
//     Enc/Inputs/In/nComState @bit 1 <-> WcState/InputToggle
//     Enc/Inputs/In/nComState <-> WcState/WcState
//     Enc/Inputs/In/nDataIn1 <-> FB Inputs Channel 1/Position
//     Enc/Inputs/In/nDataIn1 <-> FB Inputs Channel 2/Position
//     Enc/Inputs/In/nState1 @bit 12 <-> FB Inputs Channel 1/Status/Diag
//     Enc/Inputs/In/nState1 @bit 12 <-> FB Inputs Channel 2/Status/Diag
//     Enc/Inputs/In/nState1 @bit 1 <-> FB Inputs Channel 1/Status/Error
//     Enc/Inputs/In/nState1 @bit 1 <-> FB Inputs Channel 2/Status/Error
//     Enc/Inputs/In/nState1 @bit 14 <-> FB Inputs Channel 1/Status/Input cycle counter
//     Enc/Inputs/In/nState1 @bit 14 <-> FB Inputs Channel 2/Status/Input cycle counter
//     Enc/Inputs/In/nState1 @bit 2 <-> FB Inputs Channel 1/Status/Ready
//     Enc/Inputs/In/nState1 @bit 2 <-> FB Inputs Channel 2/Status/Ready
//     Enc/Inputs/In/nState1 @bit 13 <-> FB Inputs Channel 1/Status/TxPDO State
//     Enc/Inputs/In/nState1 @bit 13 <-> FB Inputs Channel 2/Status/TxPDO State
//     Enc/Inputs/In/nState1 <-> FB Inputs Channel 1/Status/Warning
//     Enc/Inputs/In/nState1 <-> FB Inputs Channel 2/Status/Warning
//   (this object) <-> HOMS/Term 1 (EK1200)/Term 2 (EK1122)/EK1100_M2L3/EL7041-1000_M2L3_PitchCoarse
//     Drive/Inputs/In/nState1 @bit 3 <-> STM Status/Status/Error
//     Drive/Inputs/In/nState1 @bit 5 <-> STM Status/Status/Moving negative
//     Drive/Inputs/In/nState1 @bit 4 <-> STM Status/Status/Moving positive
//     Drive/Inputs/In/nState1 @bit 1 <-> STM Status/Status/Ready
//     Drive/Inputs/In/nState1 <-> STM Status/Status/Ready to enable
//     Drive/Inputs/In/nState1 @bit 6 <-> STM Status/Status/Torque reduced
//     Drive/Inputs/In/nState1 @bit 2 <-> STM Status/Status/Warning
//     Drive/Inputs/In/nState2 @bit 3 <-> STM Status/Status/Digital input 1
//     Drive/Inputs/In/nState2 @bit 4 <-> STM Status/Status/Digital input 2
//     Drive/Inputs/In/nState2 @bit 5 <-> STM Status/Status/Sync error
//     Drive/Inputs/In/nState2 @bit 7 <-> STM Status/Status/TxPDO Toggle
//     Drive/Inputs/In/nState4 @bit 1 <-> WcState/InputToggle
//     Drive/Inputs/In/nState4 <-> WcState/WcState
//     Drive/Outputs/Out/nCtrl1 <-> STM Control/Control/Enable
//     Drive/Outputs/Out/nCtrl1 @bit 2 <-> STM Control/Control/Reduce torque
//     Drive/Outputs/Out/nCtrl1 @bit 1 <-> STM Control/Control/Reset
//     Drive/Outputs/Out/nDataOut2[0] <-> STM Velocity/Velocity
//   (this object) <-> HOMS/Term 1 (EK1200)/Term 2 (EK1122)/EK1100_M2L3/EL7041-1000_M2L3_Bender
//     Drive/Inputs/In/nState1 @bit 3 <-> STM Status/Status/Error
//     Drive/Inputs/In/nState1 @bit 5 <-> STM Status/Status/Moving negative
//     Drive/Inputs/In/nState1 @bit 4 <-> STM Status/Status/Moving positive
//     Drive/Inputs/In/nState1 @bit 1 <-> STM Status/Status/Ready
//     Drive/Inputs/In/nState1 <-> STM Status/Status/Ready to enable
//     Drive/Inputs/In/nState1 @bit 6 <-> STM Status/Status/Torque reduced
//     Drive/Inputs/In/nState1 @bit 2 <-> STM Status/Status/Warning
//     Drive/Inputs/In/nState2 @bit 3 <-> STM Status/Status/Digital input 1
//     Drive/Inputs/In/nState2 @bit 4 <-> STM Status/Status/Digital input 2
//     Drive/Inputs/In/nState2 @bit 5 <-> STM Status/Status/Sync error
//     Drive/Inputs/In/nState2 @bit 7 <-> STM Status/Status/TxPDO Toggle
//     Drive/Inputs/In/nState4 @bit 1 <-> WcState/InputToggle
//     Drive/Inputs/In/nState4 <-> WcState/WcState
//     Drive/Outputs/Out/nCtrl1 <-> STM Control/Control/Enable
//     Drive/Outputs/Out/nCtrl1 @bit 2 <-> STM Control/Control/Reduce torque
//     Drive/Outputs/Out/nCtrl1 @bit 1 <-> STM Control/Control/Reset
//     Drive/Outputs/Out/nDataOut2[0] <-> STM Velocity/Velocity
//   (this object) <-> HOMS/Term 1 (EK1200)/Term 14 (EK1122)/EK1100_M1L4/EL5042_M1L4_Yupdwn
//     Enc/Inputs/In/nComState @bit 1 <-> WcState/InputToggle
//     Enc/Inputs/In/nComState <-> WcState/WcState
//     Enc/Inputs/In/nDataIn1 <-> FB Inputs Channel 1/Position
//     Enc/Inputs/In/nDataIn1 <-> FB Inputs Channel 2/Position
//     Enc/Inputs/In/nState1 @bit 12 <-> FB Inputs Channel 1/Status/Diag
//     Enc/Inputs/In/nState1 @bit 12 <-> FB Inputs Channel 2/Status/Diag
//     Enc/Inputs/In/nState1 @bit 1 <-> FB Inputs Channel 1/Status/Error
//     Enc/Inputs/In/nState1 @bit 1 <-> FB Inputs Channel 2/Status/Error
//     Enc/Inputs/In/nState1 @bit 14 <-> FB Inputs Channel 1/Status/Input cycle counter
//     Enc/Inputs/In/nState1 @bit 14 <-> FB Inputs Channel 2/Status/Input cycle counter
//     Enc/Inputs/In/nState1 @bit 2 <-> FB Inputs Channel 1/Status/Ready
//     Enc/Inputs/In/nState1 @bit 2 <-> FB Inputs Channel 2/Status/Ready
//     Enc/Inputs/In/nState1 @bit 13 <-> FB Inputs Channel 1/Status/TxPDO State
//     Enc/Inputs/In/nState1 @bit 13 <-> FB Inputs Channel 2/Status/TxPDO State
//     Enc/Inputs/In/nState1 <-> FB Inputs Channel 1/Status/Warning
//     Enc/Inputs/In/nState1 <-> FB Inputs Channel 2/Status/Warning
//   (this object) <-> HOMS/Term 1 (EK1200)/Term 14 (EK1122)/EK1100_M1L4/EL7041-1000_M1L4_Yup
//     Drive/Inputs/In/nState1 @bit 3 <-> STM Status/Status/Error
//     Drive/Inputs/In/nState1 @bit 5 <-> STM Status/Status/Moving negative
//     Drive/Inputs/In/nState1 @bit 4 <-> STM Status/Status/Moving positive
//     Drive/Inputs/In/nState1 @bit 1 <-> STM Status/Status/Ready
//     Drive/Inputs/In/nState1 <-> STM Status/Status/Ready to enable
//     Drive/Inputs/In/nState1 @bit 6 <-> STM Status/Status/Torque reduced
//     Drive/Inputs/In/nState1 @bit 2 <-> STM Status/Status/Warning
//     Drive/Inputs/In/nState2 @bit 3 <-> STM Status/Status/Digital input 1
//     Drive/Inputs/In/nState2 @bit 4 <-> STM Status/Status/Digital input 2
//     Drive/Inputs/In/nState2 @bit 5 <-> STM Status/Status/Sync error
//     Drive/Inputs/In/nState2 @bit 7 <-> STM Status/Status/TxPDO Toggle
//     Drive/Inputs/In/nState4 @bit 1 <-> WcState/InputToggle
//     Drive/Inputs/In/nState4 <-> WcState/WcState
//     Drive/Outputs/Out/nCtrl1 <-> STM Control/Control/Enable
//     Drive/Outputs/Out/nCtrl1 @bit 2 <-> STM Control/Control/Reduce torque
//     Drive/Outputs/Out/nCtrl1 @bit 1 <-> STM Control/Control/Reset
//     Drive/Outputs/Out/nDataOut2[0] <-> STM Velocity/Velocity
//   (this object) <-> HOMS/Term 1 (EK1200)/Term 14 (EK1122)/EK1100_M1L4/EL7041-1000_M1L4_Ydwn
//     Drive/Inputs/In/nState1 @bit 3 <-> STM Status/Status/Error
//     Drive/Inputs/In/nState1 @bit 5 <-> STM Status/Status/Moving negative
//     Drive/Inputs/In/nState1 @bit 4 <-> STM Status/Status/Moving positive
//     Drive/Inputs/In/nState1 @bit 1 <-> STM Status/Status/Ready
//     Drive/Inputs/In/nState1 <-> STM Status/Status/Ready to enable
//     Drive/Inputs/In/nState1 @bit 6 <-> STM Status/Status/Torque reduced
//     Drive/Inputs/In/nState1 @bit 2 <-> STM Status/Status/Warning
//     Drive/Inputs/In/nState2 @bit 3 <-> STM Status/Status/Digital input 1
//     Drive/Inputs/In/nState2 @bit 4 <-> STM Status/Status/Digital input 2
//     Drive/Inputs/In/nState2 @bit 5 <-> STM Status/Status/Sync error
//     Drive/Inputs/In/nState2 @bit 7 <-> STM Status/Status/TxPDO Toggle
//     Drive/Inputs/In/nState4 @bit 1 <-> WcState/InputToggle
//     Drive/Inputs/In/nState4 <-> WcState/WcState
//     Drive/Outputs/Out/nCtrl1 <-> STM Control/Control/Enable
//     Drive/Outputs/Out/nCtrl1 @bit 2 <-> STM Control/Control/Reduce torque
//     Drive/Outputs/Out/nCtrl1 @bit 1 <-> STM Control/Control/Reset
//     Drive/Outputs/Out/nDataOut2[0] <-> STM Velocity/Velocity
//   (this object) <-> HOMS/Term 1 (EK1200)/Term 14 (EK1122)/EK1100_M1L4/EL5042_M1L4_Xupdwn
//     Enc/Inputs/In/nComState @bit 1 <-> WcState/InputToggle
//     Enc/Inputs/In/nComState <-> WcState/WcState
//     Enc/Inputs/In/nDataIn1 <-> FB Inputs Channel 1/Position
//     Enc/Inputs/In/nDataIn1 <-> FB Inputs Channel 2/Position
//     Enc/Inputs/In/nState1 @bit 12 <-> FB Inputs Channel 1/Status/Diag
//     Enc/Inputs/In/nState1 @bit 12 <-> FB Inputs Channel 2/Status/Diag
//     Enc/Inputs/In/nState1 @bit 1 <-> FB Inputs Channel 1/Status/Error
//     Enc/Inputs/In/nState1 @bit 1 <-> FB Inputs Channel 2/Status/Error
//     Enc/Inputs/In/nState1 @bit 14 <-> FB Inputs Channel 1/Status/Input cycle counter
//     Enc/Inputs/In/nState1 @bit 14 <-> FB Inputs Channel 2/Status/Input cycle counter
//     Enc/Inputs/In/nState1 @bit 2 <-> FB Inputs Channel 1/Status/Ready
//     Enc/Inputs/In/nState1 @bit 2 <-> FB Inputs Channel 2/Status/Ready
//     Enc/Inputs/In/nState1 @bit 13 <-> FB Inputs Channel 1/Status/TxPDO State
//     Enc/Inputs/In/nState1 @bit 13 <-> FB Inputs Channel 2/Status/TxPDO State
//     Enc/Inputs/In/nState1 <-> FB Inputs Channel 1/Status/Warning
//     Enc/Inputs/In/nState1 <-> FB Inputs Channel 2/Status/Warning
//   (this object) <-> HOMS/Term 1 (EK1200)/Term 14 (EK1122)/EK1100_M1L4/EL7041-1000_M1L4_Xup
//     Drive/Inputs/In/nState1 @bit 3 <-> STM Status/Status/Error
//     Drive/Inputs/In/nState1 @bit 5 <-> STM Status/Status/Moving negative
//     Drive/Inputs/In/nState1 @bit 4 <-> STM Status/Status/Moving positive
//     Drive/Inputs/In/nState1 @bit 1 <-> STM Status/Status/Ready
//     Drive/Inputs/In/nState1 <-> STM Status/Status/Ready to enable
//     Drive/Inputs/In/nState1 @bit 6 <-> STM Status/Status/Torque reduced
//     Drive/Inputs/In/nState1 @bit 2 <-> STM Status/Status/Warning
//     Drive/Inputs/In/nState2 @bit 3 <-> STM Status/Status/Digital input 1
//     Drive/Inputs/In/nState2 @bit 4 <-> STM Status/Status/Digital input 2
//     Drive/Inputs/In/nState2 @bit 5 <-> STM Status/Status/Sync error
//     Drive/Inputs/In/nState2 @bit 7 <-> STM Status/Status/TxPDO Toggle
//     Drive/Inputs/In/nState4 @bit 1 <-> WcState/InputToggle
//     Drive/Inputs/In/nState4 <-> WcState/WcState
//     Drive/Outputs/Out/nCtrl1 <-> STM Control/Control/Enable
//     Drive/Outputs/Out/nCtrl1 @bit 2 <-> STM Control/Control/Reduce torque
//     Drive/Outputs/Out/nCtrl1 @bit 1 <-> STM Control/Control/Reset
//     Drive/Outputs/Out/nDataOut2[0] <-> STM Velocity/Velocity
//   (this object) <-> HOMS/Term 1 (EK1200)/Term 14 (EK1122)/EK1100_M1L4/EL7041-1000_M1L4_Xdwn
//     Drive/Inputs/In/nState1 @bit 3 <-> STM Status/Status/Error
//     Drive/Inputs/In/nState1 @bit 5 <-> STM Status/Status/Moving negative
//     Drive/Inputs/In/nState1 @bit 4 <-> STM Status/Status/Moving positive
//     Drive/Inputs/In/nState1 @bit 1 <-> STM Status/Status/Ready
//     Drive/Inputs/In/nState1 <-> STM Status/Status/Ready to enable
//     Drive/Inputs/In/nState1 @bit 6 <-> STM Status/Status/Torque reduced
//     Drive/Inputs/In/nState1 @bit 2 <-> STM Status/Status/Warning
//     Drive/Inputs/In/nState2 @bit 3 <-> STM Status/Status/Digital input 1
//     Drive/Inputs/In/nState2 @bit 4 <-> STM Status/Status/Digital input 2
//     Drive/Inputs/In/nState2 @bit 5 <-> STM Status/Status/Sync error
//     Drive/Inputs/In/nState2 @bit 7 <-> STM Status/Status/TxPDO Toggle
//     Drive/Inputs/In/nState4 @bit 1 <-> WcState/InputToggle
//     Drive/Inputs/In/nState4 <-> WcState/WcState
//     Drive/Outputs/Out/nCtrl1 <-> STM Control/Control/Enable
//     Drive/Outputs/Out/nCtrl1 @bit 2 <-> STM Control/Control/Reduce torque
//     Drive/Outputs/Out/nCtrl1 @bit 1 <-> STM Control/Control/Reset
//     Drive/Outputs/Out/nDataOut2[0] <-> STM Velocity/Velocity
//   (this object) <-> HOMS/Term 1 (EK1200)/Term 14 (EK1122)/EK1100_M1L4/EL5042_M1L4_PitchBender
//     Enc/Inputs/In/nComState @bit 1 <-> WcState/InputToggle
//     Enc/Inputs/In/nComState <-> WcState/WcState
//     Enc/Inputs/In/nDataIn1 <-> FB Inputs Channel 1/Position
//     Enc/Inputs/In/nDataIn1 <-> FB Inputs Channel 2/Position
//     Enc/Inputs/In/nState1 @bit 12 <-> FB Inputs Channel 1/Status/Diag
//     Enc/Inputs/In/nState1 @bit 12 <-> FB Inputs Channel 2/Status/Diag
//     Enc/Inputs/In/nState1 @bit 1 <-> FB Inputs Channel 1/Status/Error
//     Enc/Inputs/In/nState1 @bit 1 <-> FB Inputs Channel 2/Status/Error
//     Enc/Inputs/In/nState1 @bit 14 <-> FB Inputs Channel 1/Status/Input cycle counter
//     Enc/Inputs/In/nState1 @bit 14 <-> FB Inputs Channel 2/Status/Input cycle counter
//     Enc/Inputs/In/nState1 @bit 2 <-> FB Inputs Channel 1/Status/Ready
//     Enc/Inputs/In/nState1 @bit 2 <-> FB Inputs Channel 2/Status/Ready
//     Enc/Inputs/In/nState1 @bit 13 <-> FB Inputs Channel 1/Status/TxPDO State
//     Enc/Inputs/In/nState1 @bit 13 <-> FB Inputs Channel 2/Status/TxPDO State
//     Enc/Inputs/In/nState1 <-> FB Inputs Channel 1/Status/Warning
//     Enc/Inputs/In/nState1 <-> FB Inputs Channel 2/Status/Warning
//   (this object) <-> HOMS/Term 1 (EK1200)/Term 14 (EK1122)/EK1100_M1L4/EL7041-1000_M1L4_PitchCoarse
//     Drive/Inputs/In/nState1 @bit 3 <-> STM Status/Status/Error
//     Drive/Inputs/In/nState1 @bit 5 <-> STM Status/Status/Moving negative
//     Drive/Inputs/In/nState1 @bit 4 <-> STM Status/Status/Moving positive
//     Drive/Inputs/In/nState1 @bit 1 <-> STM Status/Status/Ready
//     Drive/Inputs/In/nState1 <-> STM Status/Status/Ready to enable
//     Drive/Inputs/In/nState1 @bit 6 <-> STM Status/Status/Torque reduced
//     Drive/Inputs/In/nState1 @bit 2 <-> STM Status/Status/Warning
//     Drive/Inputs/In/nState2 @bit 3 <-> STM Status/Status/Digital input 1
//     Drive/Inputs/In/nState2 @bit 4 <-> STM Status/Status/Digital input 2
//     Drive/Inputs/In/nState2 @bit 5 <-> STM Status/Status/Sync error
//     Drive/Inputs/In/nState2 @bit 7 <-> STM Status/Status/TxPDO Toggle
//     Drive/Inputs/In/nState4 @bit 1 <-> WcState/InputToggle
//     Drive/Inputs/In/nState4 <-> WcState/WcState
//     Drive/Outputs/Out/nCtrl1 <-> STM Control/Control/Enable
//     Drive/Outputs/Out/nCtrl1 @bit 2 <-> STM Control/Control/Reduce torque
//     Drive/Outputs/Out/nCtrl1 @bit 1 <-> STM Control/Control/Reset
//     Drive/Outputs/Out/nDataOut2[0] <-> STM Velocity/Velocity
//   (this object) <-> HOMS/Term 1 (EK1200)/Term 14 (EK1122)/EK1100_M1L4/EL7041-1000_M1L4_Bender
//     Drive/Inputs/In/nState1 @bit 3 <-> STM Status/Status/Error
//     Drive/Inputs/In/nState1 @bit 5 <-> STM Status/Status/Moving negative
//     Drive/Inputs/In/nState1 @bit 4 <-> STM Status/Status/Moving positive
//     Drive/Inputs/In/nState1 @bit 1 <-> STM Status/Status/Ready
//     Drive/Inputs/In/nState1 <-> STM Status/Status/Ready to enable
//     Drive/Inputs/In/nState1 @bit 6 <-> STM Status/Status/Torque reduced
//     Drive/Inputs/In/nState1 @bit 2 <-> STM Status/Status/Warning
//     Drive/Inputs/In/nState2 @bit 3 <-> STM Status/Status/Digital input 1
//     Drive/Inputs/In/nState2 @bit 4 <-> STM Status/Status/Digital input 2
//     Drive/Inputs/In/nState2 @bit 5 <-> STM Status/Status/Sync error
//     Drive/Inputs/In/nState2 @bit 7 <-> STM Status/Status/TxPDO Toggle
//     Drive/Inputs/In/nState4 @bit 1 <-> WcState/InputToggle
//     Drive/Inputs/In/nState4 <-> WcState/WcState
//     Drive/Outputs/Out/nCtrl1 <-> STM Control/Control/Enable
//     Drive/Outputs/Out/nCtrl1 @bit 2 <-> STM Control/Control/Reduce torque
//     Drive/Outputs/Out/nCtrl1 @bit 1 <-> STM Control/Control/Reset
//     Drive/Outputs/Out/nDataOut2[0] <-> STM Velocity/Velocity
//   HOMS_XRT_PLC Instance <-> HOMS
//     PlcTask Inputs/GVL.gAmsNetIDEcatMaster1 <-> InfoData/AmsNetId
//   HOMS_XRT_PLC Instance <-> HOMS/Term 1 (EK1200)/Term 13 (EL2008)
//     PlcTask Outputs/GVL.bXRT_M2_IN <-> Channel 2/Output
//     PlcTask Outputs/GVL.bXRT_M2_OUT <-> Channel 1/Output
//   HOMS_XRT_PLC Instance <-> HOMS/Term 1 (EK1200)/Term 14 (EK1122)/EK1100_M1L3/EL1004_M1L3_STO
//     PlcTask Inputs/Main.MR1L3.fbRunHOMS.bSTOEnable1 <-> Channel 1/Input
//     PlcTask Inputs/Main.MR1L3.fbRunHOMS.bSTOEnable2 <-> Channel 2/Input
//   HOMS_XRT_PLC Instance <-> HOMS/Term 1 (EK1200)/Term 14 (EK1122)/EK1100_M1L3/EL5042_M1L3_PitchBender
//     PlcTask Inputs/GVL_MR1L3.MR1L3_Pitch.diEncCnt <-> FB Inputs Channel 1/Position
//     PlcTask Inputs/Main.M5.nRawEncoderULINT <-> FB Inputs Channel 1/Position
//     PlcTask Inputs/Main.M6.nRawEncoderULINT <-> FB Inputs Channel 2/Position
//   HOMS_XRT_PLC Instance <-> HOMS/Term 1 (EK1200)/Term 14 (EK1122)/EK1100_M1L3/EL5042_M1L3_Xupdwn
//     PlcTask Inputs/Main.M3.nRawEncoderULINT <-> FB Inputs Channel 1/Position
//     PlcTask Inputs/Main.MR1L3.fbRunHOMS.stXdwnEnc/Count <-> FB Inputs Channel 2/Position
//     PlcTask Inputs/Main.MR1L3.fbRunHOMS.stXupEnc/Count <-> FB Inputs Channel 1/Position
//   HOMS_XRT_PLC Instance <-> HOMS/Term 1 (EK1200)/Term 14 (EK1122)/EK1100_M1L3/EL5042_M1L3_Yupdwn
//     PlcTask Inputs/Main.M1.nRawEncoderULINT <-> FB Inputs Channel 1/Position
//     PlcTask Inputs/Main.MR1L3.fbRunHOMS.stYdwnEnc/Count <-> FB Inputs Channel 2/Position
//     PlcTask Inputs/Main.MR1L3.fbRunHOMS.stYupEnc/Count <-> FB Inputs Channel 1/Position
//   HOMS_XRT_PLC Instance <-> HOMS/Term 1 (EK1200)/Term 14 (EK1122)/EK1100_M1L3/EL6001_M1L3_PitchFine
//     SerialIO Inputs/GVL_SerialIO.Serial_stComIn_MR1L3/D[{0..21}] <-> COM Inputs/Data In {0..21}  (22 links)
//     SerialIO Inputs/GVL_SerialIO.Serial_stComIn_MR1L3/Status <-> COM Inputs/Status
//     SerialIO Outputs/GVL_SerialIO.Serial_stComOut_MR1L3/D[{0..21}] <-> COM Outputs/Data Out {0..21}  (22 links)
//   HOMS_XRT_PLC Instance <-> HOMS/Term 1 (EK1200)/Term 14 (EK1122)/EK1100_M1L3/EL7041-1000_M1L3_Bender
//     PlcTask Inputs/Main.M6.bLimitBackwardEnable <-> STM Status/Status/Digital input 2
//     PlcTask Inputs/Main.M6.bLimitForwardEnable <-> STM Status/Status/Digital input 1
//   HOMS_XRT_PLC Instance <-> HOMS/Term 1 (EK1200)/Term 14 (EK1122)/EK1100_M1L3/EL7041-1000_M1L3_PitchCoarse
//     PlcTask Inputs/Main.M5.bLimitBackwardEnable <-> STM Status/Status/Digital input 2
//     PlcTask Inputs/Main.M5.bLimitForwardEnable <-> STM Status/Status/Digital input 1
//   HOMS_XRT_PLC Instance <-> HOMS/Term 1 (EK1200)/Term 14 (EK1122)/EK1100_M1L3/EL7041-1000_M1L3_Xdwn
//     PlcTask Inputs/Main.M4.bLimitBackwardEnable <-> STM Status/Status/Digital input 2
//     PlcTask Inputs/Main.M4.bLimitForwardEnable <-> STM Status/Status/Digital input 1
//   HOMS_XRT_PLC Instance <-> HOMS/Term 1 (EK1200)/Term 14 (EK1122)/EK1100_M1L3/EL7041-1000_M1L3_Xup
//     PlcTask Inputs/Main.M3.bLimitBackwardEnable <-> STM Status/Status/Digital input 2
//     PlcTask Inputs/Main.M3.bLimitForwardEnable <-> STM Status/Status/Digital input 1
//   HOMS_XRT_PLC Instance <-> HOMS/Term 1 (EK1200)/Term 14 (EK1122)/EK1100_M1L3/EL7041-1000_M1L3_Ydwn
//     PlcTask Inputs/Main.M2.bLimitBackwardEnable <-> STM Status/Status/Digital input 2
//     PlcTask Inputs/Main.M2.bLimitForwardEnable <-> STM Status/Status/Digital input 1
//   HOMS_XRT_PLC Instance <-> HOMS/Term 1 (EK1200)/Term 14 (EK1122)/EK1100_M1L3/EL7041-1000_M1L3_Yup
//     PlcTask Inputs/Main.M1.bLimitBackwardEnable <-> STM Status/Status/Digital input 2
//     PlcTask Inputs/Main.M1.bLimitForwardEnable <-> STM Status/Status/Digital input 1
//   HOMS_XRT_PLC Instance <-> HOMS/Term 1 (EK1200)/Term 14 (EK1122)/EK1100_M1L3/MR1L3-EL3202-0010-E13
//     PlcTask Inputs/GVL_RTDS.fbMR1L3_Env_RTD_1.bError <-> RTD Inputs Channel 1/Status/Error
//     PlcTask Inputs/GVL_RTDS.fbMR1L3_Env_RTD_1.bOverrange <-> RTD Inputs Channel 1/Status/Overrange
//     PlcTask Inputs/GVL_RTDS.fbMR1L3_Env_RTD_1.bUnderrange <-> RTD Inputs Channel 1/Status/Underrange
//     PlcTask Inputs/GVL_RTDS.fbMR1L3_Env_RTD_1.iRaw <-> RTD Inputs Channel 1/Value
//   HOMS_XRT_PLC Instance <-> HOMS/Term 1 (EK1200)/Term 14 (EK1122)/EK1100_M1L3/MR1L3-EL3202-0010-E14
//     PlcTask Inputs/GVL_RTDS.fbMR1L3_Env_RTD_2.bError <-> RTD Inputs Channel 1/Status/Error
//     PlcTask Inputs/GVL_RTDS.fbMR1L3_Env_RTD_3.bError <-> RTD Inputs Channel 2/Status/Error
//     PlcTask Inputs/GVL_RTDS.fbMR1L3_Env_RTD_2.bOverrange <-> RTD Inputs Channel 1/Status/Overrange
//     PlcTask Inputs/GVL_RTDS.fbMR1L3_Env_RTD_3.bOverrange <-> RTD Inputs Channel 2/Status/Overrange
//     PlcTask Inputs/GVL_RTDS.fbMR1L3_Env_RTD_2.bUnderrange <-> RTD Inputs Channel 1/Status/Underrange
//     PlcTask Inputs/GVL_RTDS.fbMR1L3_Env_RTD_3.bUnderrange <-> RTD Inputs Channel 2/Status/Underrange
//     PlcTask Inputs/GVL_RTDS.fbMR1L3_Env_RTD_2.iRaw <-> RTD Inputs Channel 1/Value
//     PlcTask Inputs/GVL_RTDS.fbMR1L3_Env_RTD_3.iRaw <-> RTD Inputs Channel 2/Value
//   HOMS_XRT_PLC Instance <-> HOMS/Term 1 (EK1200)/Term 14 (EK1122)/EK1100_M1L4/EL1004_M1L4_STO
//     PlcTask Inputs/Main.MR1L4.fbRunHOMS.bSTOEnable1 <-> Channel 1/Input
//     PlcTask Inputs/Main.MR1L4.fbRunHOMS.bSTOEnable2 <-> Channel 2/Input
//   HOMS_XRT_PLC Instance <-> HOMS/Term 1 (EK1200)/Term 14 (EK1122)/EK1100_M1L4/EL5042_M1L4_PitchBender
//     PlcTask Inputs/GVL_MR1L4.MR1L4_Pitch.diEncCnt <-> FB Inputs Channel 1/Position
//     PlcTask Inputs/Main.M11.nRawEncoderULINT <-> FB Inputs Channel 1/Position
//     PlcTask Inputs/Main.M12.nRawEncoderULINT <-> FB Inputs Channel 2/Position
//   HOMS_XRT_PLC Instance <-> HOMS/Term 1 (EK1200)/Term 14 (EK1122)/EK1100_M1L4/EL5042_M1L4_Xupdwn
//     PlcTask Inputs/Main.M9.nRawEncoderULINT <-> FB Inputs Channel 1/Position
//     PlcTask Inputs/Main.MR1L4.fbRunHOMS.stXdwnEnc/Count <-> FB Inputs Channel 2/Position
//     PlcTask Inputs/Main.MR1L4.fbRunHOMS.stXupEnc/Count <-> FB Inputs Channel 1/Position
//   HOMS_XRT_PLC Instance <-> HOMS/Term 1 (EK1200)/Term 14 (EK1122)/EK1100_M1L4/EL5042_M1L4_Yupdwn
//     PlcTask Inputs/Main.M7.nRawEncoderULINT <-> FB Inputs Channel 1/Position
//     PlcTask Inputs/Main.MR1L4.fbRunHOMS.stYdwnEnc/Count <-> FB Inputs Channel 2/Position
//     PlcTask Inputs/Main.MR1L4.fbRunHOMS.stYupEnc/Count <-> FB Inputs Channel 1/Position
//   HOMS_XRT_PLC Instance <-> HOMS/Term 1 (EK1200)/Term 14 (EK1122)/EK1100_M1L4/EL6001_M1L4_PitchFine
//     SerialIO Inputs/GVL_SerialIO.Serial_stComIn_MR1L4/D[{0..21}] <-> COM Inputs/Data In {0..21}  (22 links)
//     SerialIO Inputs/GVL_SerialIO.Serial_stComIn_MR1L4/Status <-> COM Inputs/Status
//     SerialIO Outputs/GVL_SerialIO.Serial_stComOut_MR1L4/D[{0..21}] <-> COM Outputs/Data Out {0..21}  (22 links)
//   HOMS_XRT_PLC Instance <-> HOMS/Term 1 (EK1200)/Term 14 (EK1122)/EK1100_M1L4/EL7041-1000_M1L4_Bender
//     PlcTask Inputs/Main.M12.bLimitBackwardEnable <-> STM Status/Status/Digital input 2
//     PlcTask Inputs/Main.M12.bLimitForwardEnable <-> STM Status/Status/Digital input 1
//   HOMS_XRT_PLC Instance <-> HOMS/Term 1 (EK1200)/Term 14 (EK1122)/EK1100_M1L4/EL7041-1000_M1L4_PitchCoarse
//     PlcTask Inputs/Main.M11.bLimitBackwardEnable <-> STM Status/Status/Digital input 2
//     PlcTask Inputs/Main.M11.bLimitForwardEnable <-> STM Status/Status/Digital input 1
//   HOMS_XRT_PLC Instance <-> HOMS/Term 1 (EK1200)/Term 14 (EK1122)/EK1100_M1L4/EL7041-1000_M1L4_Xdwn
//     PlcTask Inputs/Main.M10.bLimitBackwardEnable <-> STM Status/Status/Digital input 2
//     PlcTask Inputs/Main.M10.bLimitForwardEnable <-> STM Status/Status/Digital input 1
//   HOMS_XRT_PLC Instance <-> HOMS/Term 1 (EK1200)/Term 14 (EK1122)/EK1100_M1L4/EL7041-1000_M1L4_Xup
//     PlcTask Inputs/Main.M9.bLimitBackwardEnable <-> STM Status/Status/Digital input 2
//     PlcTask Inputs/Main.M9.bLimitForwardEnable <-> STM Status/Status/Digital input 1
//   HOMS_XRT_PLC Instance <-> HOMS/Term 1 (EK1200)/Term 14 (EK1122)/EK1100_M1L4/EL7041-1000_M1L4_Ydwn
//     PlcTask Inputs/Main.M8.bLimitBackwardEnable <-> STM Status/Status/Digital input 2
//     PlcTask Inputs/Main.M8.bLimitForwardEnable <-> STM Status/Status/Digital input 1
//   HOMS_XRT_PLC Instance <-> HOMS/Term 1 (EK1200)/Term 14 (EK1122)/EK1100_M1L4/EL7041-1000_M1L4_Yup
//     PlcTask Inputs/Main.M7.bLimitBackwardEnable <-> STM Status/Status/Digital input 2
//     PlcTask Inputs/Main.M7.bLimitForwardEnable <-> STM Status/Status/Digital input 1
//   HOMS_XRT_PLC Instance <-> HOMS/Term 1 (EK1200)/Term 14 (EK1122)/EK1100_M1L4/MR1L4-EL3202-0010-E13
//     PlcTask Inputs/GVL_RTDS.fbMR1L4_Env_RTD_1.bError <-> RTD Inputs Channel 1/Status/Error
//     PlcTask Inputs/GVL_RTDS.fbMR1L4_Env_RTD_1.bOverrange <-> RTD Inputs Channel 1/Status/Overrange
//     PlcTask Inputs/GVL_RTDS.fbMR1L4_Env_RTD_1.bUnderrange <-> RTD Inputs Channel 1/Status/Underrange
//     PlcTask Inputs/GVL_RTDS.fbMR1L4_Env_RTD_1.iRaw <-> RTD Inputs Channel 1/Value
//   HOMS_XRT_PLC Instance <-> HOMS/Term 1 (EK1200)/Term 14 (EK1122)/EK1100_M1L4/MR1L4-EL3202-0010-E14
//     PlcTask Inputs/GVL_RTDS.fbMR1L4_Env_RTD_2.bError <-> RTD Inputs Channel 1/Status/Error
//     PlcTask Inputs/GVL_RTDS.fbMR1L4_Env_RTD_3.bError <-> RTD Inputs Channel 2/Status/Error
//     PlcTask Inputs/GVL_RTDS.fbMR1L4_Env_RTD_2.bOverrange <-> RTD Inputs Channel 1/Status/Overrange
//     PlcTask Inputs/GVL_RTDS.fbMR1L4_Env_RTD_3.bOverrange <-> RTD Inputs Channel 2/Status/Overrange
//     PlcTask Inputs/GVL_RTDS.fbMR1L4_Env_RTD_2.bUnderrange <-> RTD Inputs Channel 1/Status/Underrange
//     PlcTask Inputs/GVL_RTDS.fbMR1L4_Env_RTD_3.bUnderrange <-> RTD Inputs Channel 2/Status/Underrange
//     PlcTask Inputs/GVL_RTDS.fbMR1L4_Env_RTD_2.iRaw <-> RTD Inputs Channel 1/Value
//     PlcTask Inputs/GVL_RTDS.fbMR1L4_Env_RTD_3.iRaw <-> RTD Inputs Channel 2/Value
//   HOMS_XRT_PLC Instance <-> HOMS/Term 1 (EK1200)/Term 2 (EK1122)/EK1100_M2L3/EL1004_M2L3_STO
//     PlcTask Inputs/Main.MR2L3.fbRunHOMS.bSTOEnable1 <-> Channel 1/Input
//     PlcTask Inputs/Main.MR2L3.fbRunHOMS.bSTOEnable2 <-> Channel 2/Input
//   HOMS_XRT_PLC Instance <-> HOMS/Term 1 (EK1200)/Term 2 (EK1122)/EK1100_M2L3/EL5042_M2L3_PitchBender
//     PlcTask Inputs/Main.M17.nRawEncoderULINT <-> FB Inputs Channel 1/Position
//     PlcTask Inputs/Main.M18.nRawEncoderULINT <-> FB Inputs Channel 2/Position
//   HOMS_XRT_PLC Instance <-> HOMS/Term 1 (EK1200)/Term 2 (EK1122)/EK1100_M2L3/EL5042_M2L3_Xupdwn
//     PlcTask Inputs/Main.M15.nRawEncoderULINT <-> FB Inputs Channel 1/Position
//     PlcTask Inputs/Main.MR2L3.fbRunHOMS.stXdwnEnc/Count <-> FB Inputs Channel 2/Position
//     PlcTask Inputs/Main.MR2L3.fbRunHOMS.stXupEnc/Count <-> FB Inputs Channel 1/Position
//   HOMS_XRT_PLC Instance <-> HOMS/Term 1 (EK1200)/Term 2 (EK1122)/EK1100_M2L3/EL5042_M2L3_Yupdwn
//     PlcTask Inputs/Main.MR2L3.fbRunHOMS.stYdwnEnc/Count <-> FB Inputs Channel 2/Position
//     PlcTask Inputs/Main.MR2L3.fbRunHOMS.stYupEnc/Count <-> FB Inputs Channel 1/Position
//   HOMS_XRT_PLC Instance <-> HOMS/Term 1 (EK1200)/Term 2 (EK1122)/EK1100_M2L3/EL6001_M2L3_PitchFine
//     SerialIO Inputs/GVL_SerialIO.Serial_stComIn_MR2L3/D[{0..21}] <-> COM Inputs/Data In {0..21}  (22 links)
//     SerialIO Inputs/GVL_SerialIO.Serial_stComIn_MR2L3/Status <-> COM Inputs/Status
//     SerialIO Outputs/GVL_SerialIO.Serial_stComOut_MR2L3/D[{0..21}] <-> COM Outputs/Data Out {0..21}  (22 links)
//   HOMS_XRT_PLC Instance <-> HOMS/Term 1 (EK1200)/Term 2 (EK1122)/EK1100_M2L3/EL7041-1000_M2L3_Bender
//     PlcTask Inputs/Main.M18.bLimitBackwardEnable <-> STM Status/Status/Digital input 2
//     PlcTask Inputs/Main.M18.bLimitForwardEnable <-> STM Status/Status/Digital input 1
//   HOMS_XRT_PLC Instance <-> HOMS/Term 1 (EK1200)/Term 2 (EK1122)/EK1100_M2L3/EL7041-1000_M2L3_PitchCoarse
//     PlcTask Inputs/Main.M17.bLimitBackwardEnable <-> STM Status/Status/Digital input 2
//     PlcTask Inputs/Main.M17.bLimitForwardEnable <-> STM Status/Status/Digital input 1
//   HOMS_XRT_PLC Instance <-> HOMS/Term 1 (EK1200)/Term 2 (EK1122)/EK1100_M2L3/EL7041-1000_M2L3_Xdwn
//     PlcTask Inputs/Main.M16.bLimitBackwardEnable <-> STM Status/Status/Digital input 2
//     PlcTask Inputs/Main.M16.bLimitForwardEnable <-> STM Status/Status/Digital input 1
//   HOMS_XRT_PLC Instance <-> HOMS/Term 1 (EK1200)/Term 2 (EK1122)/EK1100_M2L3/EL7041-1000_M2L3_Xup
//     PlcTask Inputs/Main.M15.bLimitBackwardEnable <-> STM Status/Status/Digital input 2
//     PlcTask Inputs/Main.M15.bLimitForwardEnable <-> STM Status/Status/Digital input 1
//   HOMS_XRT_PLC Instance <-> HOMS/Term 1 (EK1200)/Term 2 (EK1122)/EK1100_M2L3/EL7041-1000_M2L3_Ydwn
//     PlcTask Inputs/Main.M14.bLimitBackwardEnable <-> STM Status/Status/Digital input 2
//     PlcTask Inputs/Main.M14.bLimitForwardEnable <-> STM Status/Status/Digital input 1
//   HOMS_XRT_PLC Instance <-> HOMS/Term 1 (EK1200)/Term 2 (EK1122)/EK1100_M2L3/EL7041-1000_M2L3_Yup
//     PlcTask Inputs/Main.M13.bLimitBackwardEnable <-> STM Status/Status/Digital input 2
//     PlcTask Inputs/Main.M13.bLimitForwardEnable <-> STM Status/Status/Digital input 1
//   HOMS_XRT_PLC Instance <-> HOMS/Term 1 (EK1200)/Term 2 (EK1122)/EK1100_M2L3/MR2L3-EL3202-0010-E13
//     PlcTask Inputs/GVL_RTDS.fbMR2L3_Env_RTD_1.bError <-> RTD Inputs Channel 1/Status/Error
//     PlcTask Inputs/GVL_RTDS.fbMR2L3_Env_RTD_1.bOverrange <-> RTD Inputs Channel 1/Status/Overrange
//     PlcTask Inputs/GVL_RTDS.fbMR2L3_Env_RTD_1.bUnderrange <-> RTD Inputs Channel 1/Status/Underrange
//     PlcTask Inputs/GVL_RTDS.fbMR2L3_Env_RTD_1.iRaw <-> RTD Inputs Channel 1/Value
//   HOMS_XRT_PLC Instance <-> HOMS/Term 1 (EK1200)/Term 2 (EK1122)/EK1100_M2L3/MR2L3-EL3202-0010-E14
//     PlcTask Inputs/GVL_RTDS.fbMR2L3_Env_RTD_2.bError <-> RTD Inputs Channel 1/Status/Error
//     PlcTask Inputs/GVL_RTDS.fbMR2L3_Env_RTD_3.bError <-> RTD Inputs Channel 2/Status/Error
//     PlcTask Inputs/GVL_RTDS.fbMR2L3_Env_RTD_2.bOverrange <-> RTD Inputs Channel 1/Status/Overrange
//     PlcTask Inputs/GVL_RTDS.fbMR2L3_Env_RTD_3.bOverrange <-> RTD Inputs Channel 2/Status/Overrange
//     PlcTask Inputs/GVL_RTDS.fbMR2L3_Env_RTD_2.bUnderrange <-> RTD Inputs Channel 1/Status/Underrange
//     PlcTask Inputs/GVL_RTDS.fbMR2L3_Env_RTD_3.bUnderrange <-> RTD Inputs Channel 2/Status/Underrange
//     PlcTask Inputs/GVL_RTDS.fbMR2L3_Env_RTD_2.iRaw <-> RTD Inputs Channel 1/Value
//     PlcTask Inputs/GVL_RTDS.fbMR2L3_Env_RTD_3.iRaw <-> RTD Inputs Channel 2/Value
//   HOMS_XRT_PLC Instance <-> HOMS/Term 1 (EK1200)/Term 34 (EK1521-0010)/Term 23 (EK1501-0010)/PMPS_FFO
//     PlcTask Outputs/GVL_PMPS.g_FastFaultOutput1.q_xFastFaultOut <-> Channel 1/Output
//     PlcTask Outputs/GVL_PMPS.g_FastFaultOutput2.q_xFastFaultOut <-> Channel 2/Output
//   HOMS_XRT_PLC Instance <-> HOMS/Term 1 (EK1200)/Term 34 (EK1521-0010)/Term 23 (EK1501-0010)/PMPS_PRE
//     PlcTask Inputs/GVL_PMPS.fbArbiterIO.i_stCurrentBP <-> IO Inputs/CurrentBP
//     PlcTask Inputs/GVL_PMPS.fbArbiterIO.xTxPDO_state <-> SYNC Inputs/TxPDO state
//     PlcTask Inputs/GVL_PMPS.fbArbiterIO.xTxPDO_toggle <-> SYNC Inputs/TxPDO toggle
//     PlcTask Outputs/GVL_PMPS.fbArbiterIO.q_stRequestedBP <-> IO Outputs/RequestedBP
//   HOMS_XRT_PLC Instance <-> NC-Task 1 SAF/Axes/M1L3-Bender
//     PlcTask Inputs/Main.M6.Axis.NcToPlc <-> Outputs/ToPlc
//     PlcTask Outputs/Main.M6.Axis.PlcToNc <-> Inputs/FromPlc
//   HOMS_XRT_PLC Instance <-> NC-Task 1 SAF/Axes/M1L3-Pitch
//     PlcTask Inputs/Main.M5.Axis.NcToPlc <-> Outputs/ToPlc
//     PlcTask Outputs/Main.M5.Axis.PlcToNc <-> Inputs/FromPlc
//   HOMS_XRT_PLC Instance <-> NC-Task 1 SAF/Axes/M1L3-Xdwn
//     PlcTask Inputs/Main.M4.Axis.NcToPlc <-> Outputs/ToPlc
//     PlcTask Outputs/Main.M4.Axis.PlcToNc <-> Inputs/FromPlc
//   HOMS_XRT_PLC Instance <-> NC-Task 1 SAF/Axes/M1L3-Xup
//     PlcTask Inputs/Main.M3.Axis.NcToPlc <-> Outputs/ToPlc
//     PlcTask Outputs/Main.M3.Axis.PlcToNc <-> Inputs/FromPlc
//   HOMS_XRT_PLC Instance <-> NC-Task 1 SAF/Axes/M1L3-Ydwn
//     PlcTask Inputs/Main.M2.Axis.NcToPlc <-> Outputs/ToPlc
//     PlcTask Outputs/Main.M2.Axis.PlcToNc <-> Inputs/FromPlc
//   HOMS_XRT_PLC Instance <-> NC-Task 1 SAF/Axes/M1L3-Yup
//     PlcTask Inputs/Main.M1.Axis.NcToPlc <-> Outputs/ToPlc
//     PlcTask Outputs/Main.M1.Axis.PlcToNc <-> Inputs/FromPlc
//   HOMS_XRT_PLC Instance <-> NC-Task 1 SAF/Axes/M1L4-Bender
//     PlcTask Inputs/Main.M12.Axis.NcToPlc <-> Outputs/ToPlc
//     PlcTask Outputs/Main.M12.Axis.PlcToNc <-> Inputs/FromPlc
//   HOMS_XRT_PLC Instance <-> NC-Task 1 SAF/Axes/M1L4-Pitch
//     PlcTask Inputs/Main.M11.Axis.NcToPlc <-> Outputs/ToPlc
//     PlcTask Outputs/Main.M11.Axis.PlcToNc <-> Inputs/FromPlc
//   HOMS_XRT_PLC Instance <-> NC-Task 1 SAF/Axes/M1L4-Xdwn
//     PlcTask Inputs/Main.M10.Axis.NcToPlc <-> Outputs/ToPlc
//     PlcTask Outputs/Main.M10.Axis.PlcToNc <-> Inputs/FromPlc
//   HOMS_XRT_PLC Instance <-> NC-Task 1 SAF/Axes/M1L4-Xup
//     PlcTask Inputs/Main.M9.Axis.NcToPlc <-> Outputs/ToPlc
//     PlcTask Outputs/Main.M9.Axis.PlcToNc <-> Inputs/FromPlc
//   HOMS_XRT_PLC Instance <-> NC-Task 1 SAF/Axes/M1L4-Ydwn
//     PlcTask Inputs/Main.M8.Axis.NcToPlc <-> Outputs/ToPlc
//     PlcTask Outputs/Main.M8.Axis.PlcToNc <-> Inputs/FromPlc
//   HOMS_XRT_PLC Instance <-> NC-Task 1 SAF/Axes/M1L4-Yup
//     PlcTask Inputs/Main.M7.Axis.NcToPlc <-> Outputs/ToPlc
//     PlcTask Outputs/Main.M7.Axis.PlcToNc <-> Inputs/FromPlc
//   HOMS_XRT_PLC Instance <-> NC-Task 1 SAF/Axes/M2L3-Bender
//     PlcTask Inputs/Main.M18.Axis.NcToPlc <-> Outputs/ToPlc
//     PlcTask Outputs/Main.M18.Axis.PlcToNc <-> Inputs/FromPlc
//   HOMS_XRT_PLC Instance <-> NC-Task 1 SAF/Axes/M2L3-Pitch
//     PlcTask Inputs/Main.M17.Axis.NcToPlc <-> Outputs/ToPlc
//     PlcTask Outputs/Main.M17.Axis.PlcToNc <-> Inputs/FromPlc
//   HOMS_XRT_PLC Instance <-> NC-Task 1 SAF/Axes/M2L3-Xdwn
//     PlcTask Inputs/Main.M16.Axis.NcToPlc <-> Outputs/ToPlc
//     PlcTask Outputs/Main.M16.Axis.PlcToNc <-> Inputs/FromPlc
//   HOMS_XRT_PLC Instance <-> NC-Task 1 SAF/Axes/M2L3-Xup
//     PlcTask Inputs/Main.M15.Axis.NcToPlc <-> Outputs/ToPlc
//     PlcTask Outputs/Main.M15.Axis.PlcToNc <-> Inputs/FromPlc
//   HOMS_XRT_PLC Instance <-> NC-Task 1 SAF/Axes/M2L3-Ydwn
//     PlcTask Inputs/Main.M14.Axis.NcToPlc <-> Outputs/ToPlc
//     PlcTask Outputs/Main.M14.Axis.PlcToNc <-> Inputs/FromPlc
//   HOMS_XRT_PLC Instance <-> NC-Task 1 SAF/Axes/M2L3-Yup
//     PlcTask Inputs/Main.M13.Axis.NcToPlc <-> Outputs/ToPlc
//     PlcTask Outputs/Main.M13.Axis.PlcToNc <-> Inputs/FromPlc

CONFIGURATION HOMS_XRT_PLC
    RESOURCE PLC ON TwinCAT3
        TASK PiezoDriver(INTERVAL := T#1ms, PRIORITY := 3);
        TASK PlcTask(INTERVAL := T#10ms, PRIORITY := 20);
        TASK SerialIO(INTERVAL := T#2ms, PRIORITY := 1);
        PROGRAM PiezoSerial WITH PiezoDriver : PiezoSerial;
        PROGRAM P_Serial_Com WITH SerialIO : P_Serial_Com;
    END_RESOURCE
END_CONFIGURATION

// ---- Common/DUTs/ENUM_Coating_States.TcDUT
{attribute 'qualified only'}
TYPE ENUM_Coating_States :
(
    Unknown := 0,
    SiC := 1,
    W := 2
);
END_TYPE

// ---- Common/DUTs/E_GantryControl.TcDUT
TYPE E_GantryControl :
(
    //Gantry Control Machine
    GCM_Idle := 0,
    GCM_Init := 5,
    GCM_ChangeCoupling := 10,
    GCM_Couple := 50,
    GCM_CoupledEnable := 51,
    GCM_CoupledStandby := 100,
    GCM_Decouple := 500,
    GCM_DecoupledStandby := 1000,
    GCM_CoupledMoveDone	:= 8000,
    GCM_Error	:= 9000
);
END_TYPE

// ---- Common/DUTs/E_GantryMode.TcDUT
TYPE E_GantryMode :
(
    GantryModeCoupled := 0,
    GantryModeDecoupled	:= 1
);
END_TYPE

// ---- Common/DUTs/E_PiezoControl.TcDUT
TYPE E_PiezoControl :
(
    //Piezo Control Machine
    EPC_Idle := 0,
    EPC_Init := 10,
    EPC_MoveRequested  := 50,
    EPC_MovingPositive := 100,
    EPC_MovingNegative := 200,
    EPC_MoveCompleted  := 350,
    EPC_Error := 500
);
END_TYPE

// ---- Common/DUTs/E_PitchControl.TcDUT
TYPE E_PitchControl :
(
    //Pitch Control Machine
    PCM_Init := 0,
    PCM_Standby := 1,
    PCM_MoveRequested := 10,
    PCM_Coarse50Piezo	:= 20,
    PCM_CoarseMove	:= 21,
    PCM_CoarseMoveCleanup := 22,
    PCM_FineMove	:= 30,
    PCM_Halt		:= 50,
    PCM_Done	:= 8000, //why is 8000 done? Where did this come from??
    PCM_Error   := 9000, //Anything above 9000 is considered an error
    PCM_StepperError	:= 9100,
    PCM_PiezoError	:= 9200,
    PCM_OtherError := 9300
);
END_TYPE

// ---- Common/DUTs/HOMS_Gantry.TcDUT
TYPE HOMS_Gantry :
STRUCT
    PAxis	:	HOMS_GantryAxis; //Primary Axis, upstream
    SAxis	:	HOMS_GantryAxis; //Secondary Axis, downstream
    VAxis	:	HOMS_GantryAxis; //Virtual Axis
    Mode	:	E_GantryMode; //Current gantry mode
    ModeReq:	E_GantryMode := GantryModeCoupled; //Requested gantry mode
    Diff	:	REAL;	//Gantry difference
    DiffFlt	:	BOOL := TRUE; //Gantry difference fault, true means fault
    xCoupled : BOOL := FALSE;
    xUncouple   : BOOL := FALSE;//Switch to uncouple axis
    PAxisActPos	:	LREAL; //Encoder Readback
    SAxisActPos	:	LREAL; //Encoder Readback

    (* Parameters
    These should come primarily from the ESD *)
    DiffTol	:	LREAL := 0.200;	//Gantry difference tolerance (mm)
    DiffHys	:	LREAL := 0.050;	//Gantry difference hysteresis (mm)
END_STRUCT
END_TYPE

// ---- Common/DUTs/HOMS_GantryAxis.TcDUT
TYPE HOMS_GantryAxis EXTENDS ST_HOMSStepper :
STRUCT
    //Virtual limit switch derived from gantry difference
    DecoupledPositiveEnable	:	BOOL;
    DecoupledNegativeEnable	:	BOOL;

    //Axis center as defined in Axilon FAT, used for gantry difference calculation adjustment
    cCenter	:	DINT := 0;

    //Raw encoder count
    diEncCnt	AT %I*	:	DINT;

END_STRUCT
END_TYPE

// ---- Common/DUTs/HOMS_PitchMechanismOld.TcDUT
TYPE HOMS_PitchMechanismOld :
STRUCT
    Piezo	:	ST_PiezoAxisOld;	//Piezo
    Axis	:	ST_AbstractAxis; //Abstract pitch axis
    Stepper	:	ST_HOMSStepper; //Pitch stepper axis

    (* Soft limits, egu urad *)
    ReqPosLimHi	:	REAL;
    ReqPosLimLo	:	REAL;


    (* Hard limits, egu INC *)
    (* These are discovered during installation, and represent encoder ticks, unbiased *)
    (* We changed to these when our pitch mechanism limit switches were insufficient for
    good control. They had too much hysteresis/ lack of precision. At this point the limit
    switches are ignored, and instead their function is carried out by these. *)
    diEncPosLimHi	:	DINT;
    diEncPosLimLo	:	DINT;
    //Raw encoder count
    diEncCnt	AT %I*	:	DINT;


END_STRUCT
END_TYPE

// ---- Common/DUTs/ST_AbstractAxis.TcDUT
TYPE ST_AbstractAxis :
STRUCT
(* ST_BasicAxis was created for basic motion controls. AbstractAxis
is similar, but removes some unused elements that don't apply to axes
that are not directly linked to hardware, eg. axes that are combinations
of more than one physical actuator. *)

(* Controls *)
xEnable	:	BOOL;
rReqAbsPos	:	REAL;
lrVelocity	:	REAL	:=1; //mm/s
xStartAbsMove	:	BOOL;
xStop	:	BOOL;
xReset	:	BOOL;
//Tweak Requests
bTwkFwd : BOOL;
bTwkBwd : BOOL;
rTweak  : REAL;
//External motor interlock, overrides axis enable
i_xMotorInterlock	:	BOOL := FALSE;

xHiLS	:	BOOL;
xLoLS	:	BOOL;

(* Status *)
bBusy 	:	BOOL;
bDone 	:	BOOL;

END_STRUCT
END_TYPE

// ---- Common/DUTs/ST_CoEIndSub.TcDUT
TYPE ST_CoEIndSub :
STRUCT
    nIndex	:	WORD;
    nSubIndex	:	BYTE;
END_STRUCT
END_TYPE

// ---- Common/DUTs/ST_DecoupledMotionPermits.TcDUT
TYPE ST_DecoupledMotionPermits :
STRUCT
    // Positive direction permit in decoupled mode
    Positive	:	BOOL;
    // Negative direction permit in decoupled mode
    Negative	:	BOOL;
END_STRUCT
END_TYPE

// ---- Common/DUTs/ST_ElmoGDCBellCoEParams.TcDUT
TYPE ST_ElmoGDCBellCoEParams :
STRUCT
        //Drive Reference (for CoE)
        stDriveRef	 :	ST_DriveRef; //Note, ignore the ams id and type parameters for our purposes.
        //Ams id comes from a linked global variable
        stPlcDriveRef AT %I* : ST_PlcDriveRef;

        AmsID	:	T_AmsNetId;
        nSlave	:	UINT;

        //Additional drive parameters
        //5V supply for encoders/ misc
        ui5VSupply :	UINT;
        //Drive temperature, C
        uiDriveTemp	:	UINT;

        // Checksum
        testChecksum : DINT;
END_STRUCT
END_TYPE

// ---- Common/DUTs/ST_HOMSStepper.TcDUT
TYPE ST_HOMSStepper :
STRUCT

    (* Controls *)
    /////////////////////////////////
    xEnable	:	BOOL;
    xReset	:	BOOL;
    //External motor interlock, overrides axis enable
    i_xMotorInterlock	:	BOOL;
    //Motion Profile
    fVelocity     : REAL;
    fAcceleration : REAL;
    fDeceleration : REAL ;
    //Tweak Requests
    bTwkFwd : BOOL;
    bTwkBwd : BOOL;
    rTweak  : REAL;
    //Absolute Value Request
    rReqAbsolute : REAL:= 0.0;
    //Pitch stepper dmov range (urad)
    rStepperDmovRange	:	REAL := 20;
    (* Status *)
    //Axis Status
    stStatus : ST_StepperStatus;
    bDone : BOOL;
    bBusy : BOOL;


    (* IO *)
    //CoE Stuff
    ///////////////////////////////
    stCoE	:	ST_ElmoGDCBellCoEParams;

    //Drive inputs
    /////////////////////////////
    diInputs	AT %I*	:	DINT;
    //Drive current
    iDriveCurrent	AT %I*	:	INT;
    (* Axis motor *)
    stAxis	:	AXIS_REF;
    //Limit switches
    xHiLS	:	BOOL;
    xLoLS	:	BOOL;



END_STRUCT
END_TYPE

// ---- Common/DUTs/ST_PiezoAxisOld.TcDUT
TYPE ST_PiezoAxisOld :
STRUCT
    (* IO *)
        //Readback
        sIdn				:	STRING; //Identity
        iCurError			:	INT; //Current error code, should be 0 most of the time
        iLastError			:	INT; //Last error code, for history
        rActVoltage			:	REAL; //Actual voltage
        rLastReqVoltage		:	REAL; //Last requested piezo voltage
        //Control
        rSetVoltage			:	REAL; //this parameter is set by the control loop/ voltage mode
        sAxis				:   STRING :='A'; //Axis, e.g. A, B, C...A if single unit
        //Summaries
        xTimeout	:	BOOL;
        xDriverError		:	BOOL; //Summary of any driver errors

    (* Operation *)
        xEnable	:	BOOL; //Enable control.
        (* Note: Voltage mode and Idle mode overrides "DirectPiezoMode" of FB_PitchControl *)
        xVoltageMode	:	BOOL; //Voltage mode gives direct access to piezo voltage, false means closed loop position acquisition (see FB_PitchControl for piezo and stepper separation)
        xIdleMode	:	BOOL; //Use to put the piezo at half-stroke
        rReqVoltage : REAL; //Requested piezo voltage in voltage mode
        rReqAbsPos	:	LREAL; //Requested Position, latched at rising StartAbsMov
        xStop	:	BOOL;	//Stops piezo and holds position


    (* Control Parameters *)
        rActPos	:	LREAL; //Encoder Readback
        //Pitch piezo dmove range (urad)
        rPiezoDmovRange		:	REAL := 1;
        stPIParams	:	ST_CTRL_PI_PARAMS := (
            tCtrlCycleTime := T#0MS,
            tTaskCycleTime := T#0MS,
            tTn       := T#1S,
            fKp      := 0.25,
            fOutMaxLimit := 1,
            fOutMinLimit := -1,
            bARWOnIPartOnly := FALSE);

    (* Voltage ranges, come from specifications of the driver *)
        UpperVoltage	:	REAL := cPiezoMaxVoltage; // E-816 has no software limits
        LowerVoltage	:	REAL := cPiezoMinVoltage; // E-816 has no software limits
END_STRUCT
END_TYPE

// ---- Common/DUTs/ST_StepperStatus.TcDUT
TYPE ST_StepperStatus :
STRUCT
    bEnable: BOOL;
    bReset: BOOL;
    bExecute: BOOL;
    nCommand: UINT;
    nCmdData: UINT;
    fVelocity: LREAL;
    fPosition: REAL;
    fAcceleration: LREAL;
    fDeceleration: LREAL;
    bJogFwd: BOOL;
    bJogBwd: BOOL;
    bLimitFwd: BOOL;
    bLimitBwd: BOOL;
    fOverride: LREAL := 100;
    bHomeSensor: BOOL;
    bEnabled: BOOL;
    bError: BOOL;
    nErrorId: UDINT;
    fActVelocity: LREAL;
    fActPosition: LREAL;
    rActPosition: REAL;
    rActVelocity: REAL;
    fActDiff: LREAL;
    bHomed:BOOL;
    bBusy:BOOL;
END_STRUCT
END_TYPE

// ---- Version/Global_Version.TcGVL
{attribute 'TcGenerated'}
{attribute 'no-analysis'}
{attribute 'linkalways'}
// This function has been automatically generated from the project information.
VAR_GLOBAL CONSTANT
    {attribute 'const_non_replaced'}
    stLibVersion_lcls_plc_xrt_optics : ST_LibVersion := (iMajor := 5, iMinor := 7, iBuild := 0, iRevision := 0, nFlags := 1, sVersion := '5.7.0');
END_VAR

// ---- GVLs/GVL.TcGVL
VAR_GLOBAL
    g_psLogHost	: T_IPv4Addr := '172.21.32.9';
    gDefaultSubsystem : E_Subsystem := MOTION;
    gSystemFault	:	BOOL;
    gAmsNetIDEcatMaster1	AT %I* 	: AMSNETID;
    gFirstPass	:	 BOOL := TRUE;

    //MPS Outputs
    {attribute 'pytmc' := '
        pv: PLC:XRT:OPTICS:M2:OUT
    '}
    bXRT_M2_OUT AT %Q* : BOOL:= FALSE;
    {attribute 'pytmc' := '
        pv: PLC:XRT:OPTICS:M2:IN
    '}
    bXRT_M2_IN AT %Q* : BOOL:= FALSE;

    //Safe-torque-off status
    gM1STO	:	BOOL;
    gM2STO	:	BOOL;
    gM3STO	:	BOOL;

    //Global encoder scale
    // For the HOMS, the encoders are all 1nm/cnt which makes things very easy
    gEncScale	:	LREAL := 1;

    //Overrides
    ////////////////////////////////////
        (* Use at your own risk. These variables may induce unexpected state machine cases,
            and other undesirable effects. They are primarily for testing purposes. Do
        not use them for operations except in the most dire of situations, and with
        full knowledge and understanding of what they do. *)
        gBypassVirtualLimits	:	BOOL;

END_VAR

// ---- GVLs/GVL_COM_Buffers.TcGVL
VAR_GLOBAL

    // M1
    Serial_RXBuffer_MR1L3 : ComBuffer;
    Serial_TXBuffer_MR1L3 : ComBuffer;

    Serial_RXBuffer_MR1L4 : ComBuffer;
    Serial_TXBuffer_MR1L4 : ComBuffer;

    Serial_RXBuffer_MR2L3 : ComBuffer;
    Serial_TXBuffer_MR2L3 : ComBuffer;


END_VAR

// ---- GVLs/GVL_Constants.TcGVL
VAR_GLOBAL CONSTANT

    cPiezoMaxVoltage	:	LREAL := 120;
    cPiezoMinVoltage	:	LREAL := -10;
(*
    //FEE-M1
    ///////////////////////////
    //X
    HOMS1_XGantry_PAxisCenter : DINT:=24432540;
    HOMS1_XGantry_SAxisCenter : DINT:=25259170;

    //Y
    HOMS1_YGantry_PAxisCenter : DINT:=14890432;
    HOMS1_YGantry_SAxisCenter : DINT:=14845283;

    //FEE-M2
    ///////////////////////////
    //X
    HOMS2_XGantry_PAxisCenter : DINT:=24432540;
    HOMS2_XGantry_SAxisCenter : DINT:=25259170;

    //Y
    HOMS2_YGantry_PAxisCenter : DINT:=14890432;
    HOMS2_YGantry_SAxisCenter : DINT:=14845283;

    *)
END_VAR

// ---- GVLs/GVL_MR1L3.TcGVL
{attribute 'qualified_only'}
VAR_GLOBAL
    // Pitch Mechanism:
    {attribute 'TcLinkTo' := '.diEncCnt:=TIIB[EL5042_M1L3_PitchBender]^FB Inputs Channel 1^Position'}
    MR1L3_Pitch : HOMS_PitchMechanism := (ReqPosLimHi := 220,
                                         ReqPosLimLo := -193.0,
                                         diEncPosLimHi := 11216281,
                                         diEncPosLimLo := 11004512);
END_VAR

// ---- GVLs/GVL_MR1L4_Constants.TcGVL
{attribute 'qualified_only'}
VAR_GLOBAL CONSTANT
    // Encoder reference values in counts = nm
    // Enc Ref Vals from alignment 2020-6-12
    nYUP_ENC_REF : ULINT := 13663400;
    nYDWN_ENC_REF : ULINT := 15043000;
    nXUP_ENC_REF : ULINT := 25569700;
    nXDWN_ENC_REF : ULINT := 26702800;
END_VAR

// ---- GVLs/GVL_MR1L4.TcGVL
{attribute 'qualified_only'}
VAR_GLOBAL
    // Pitch Mechanism:
    {attribute 'TcLinkTo' := '.diEncCnt:=TIIB[EL5042_M1L4_PitchBender]^FB Inputs Channel 1^Position'}
    MR1L4_Pitch : HOMS_PitchMechanism := (ReqPosLimHi := 246,
                                         ReqPosLimLo := -212.0,
                                         diEncPosLimHi := 9951420,
                                         diEncPosLimLo := 9716400);
END_VAR

// ---- GVLs/GVL_MR1L3_Constants.TcGVL
{attribute 'qualified_only'}
VAR_GLOBAL CONSTANT
    // Encoder reference values in counts = nm
    // Enc Ref Vals from alignment 2020-6-12
    nYUP_ENC_REF : ULINT := 13611000;
    nYDWN_ENC_REF : ULINT := 13433600;
    nXUP_ENC_REF : ULINT := 25210500;
    nXDWN_ENC_REF : ULINT := 24971800;
END_VAR

// ---- GVLs/GVL_MR2L3_Constants.TcGVL
{attribute 'qualified_only'}
VAR_GLOBAL CONSTANT
    // Encoder reference values in counts = nm
    // Enc Ref Vals from alignment 2020-6-12
    nYUP_ENC_REF : ULINT := 14279350;
    nYDWN_ENC_REF : ULINT := 16316457;
    nXUP_ENC_REF : ULINT := 25135760;
    nXDWN_ENC_REF : ULINT := 24091270;
END_VAR

// ---- GVLs/GVL_MR2L3.TcGVL
{attribute 'qualified_only'}
VAR_GLOBAL
    // Pitch Mechanism:
    {attribute 'TcLinkTo' := '.diEncCnt:=TIIB[EL5042_M1_PitchBender]^FB Inputs Channel 1^Position'}
    MR2L3_Pitch : HOMS_PitchMechanism := (ReqPosLimHi := 246,
                                         ReqPosLimLo := -212.0,
                                         diEncPosLimHi := 10349000,
                                         diEncPosLimLo := 9349000);
END_VAR

// ---- GVLs/GVL_PMPS.TcGVL


{attribute 'qualified_only'}
VAR_GLOBAL
    {attribute 'pytmc' := '
    pv: PLC:XRT:OPTICS:FFO:01
    '}
    {attribute 'TcLinkTo' := '.q_xFastFaultOut:=TIIB[PMPS_FFO]^Channel 1^Output'}
    g_FastFaultOutput1  :   FB_HardwareFFOutput := (i_sNetID:='172.21.88.66.1.1');

    {attribute 'pytmc' := '
    pv: PLC:XRT:OPTICS:FFO:02
    '}
    {attribute 'TcLinkTo' := '.q_xFastFaultOut:=TIIB[PMPS_FFO]^Channel 2^Output'}
    g_FastFaultOutput2  :   FB_HardwareFFOutput := (i_sNetID:='172.21.88.66.1.1');

    {attribute 'pytmc' := '
    pv: PLC:XRT:OPTICS:ARB:01
    '}
    g_fbArbiter1 : FB_Arbiter(1);

    {attribute 'pytmc' := '
    pv: PLC:XRT:OPTICS:ARB:02
    '}
    g_fbArbiter2 : FB_Arbiter(2);

    // PMPS arbiter interface
    fbArbiterIO : FB_SubSysToArbiter_IO;

END_VAR

// ---- GVLs/GVL_RTDS.TcGVL
{attribute 'qualified_only'}
VAR_GLOBAL
    // MR1L3 RTDs
    {attribute 'TcLinkTo' := '.iRaw := TIIB[MR1L3-EL3202-0010-E13]^RTD Inputs Channel 1^Value;
                              .bUnderrange := TIIB[MR1L3-EL3202-0010-E13]^RTD Inputs Channel 1^Status^Underrange;
                              .bOverrange := TIIB[MR1L3-EL3202-0010-E13]^RTD Inputs Channel 1^Status^Overrange;
                              .bError := TIIB[MR1L3-EL3202-0010-E13]^RTD Inputs Channel 1^Status^Error'}
    {attribute 'pytmc' := '
        pv: MR1L3:HOMS:ENV:RTD:1
        field: EGU C
        io: i
    '}
    fbMR1L3_Env_RTD_1 : FB_TempSensor;
    {attribute 'TcLinkTo' := '.iRaw := TIIB[MR1L3-EL3202-0010-E14]^RTD Inputs Channel 1^Value;
                              .bUnderrange := TIIB[MR1L3-EL3202-0010-E14]^RTD Inputs Channel 1^Status^Underrange;
                              .bOverrange := TIIB[MR1L3-EL3202-0010-E14]^RTD Inputs Channel 1^Status^Overrange;
                              .bError := TIIB[MR1L3-EL3202-0010-E14]^RTD Inputs Channel 1^Status^Error'}
    {attribute 'pytmc' := '
        pv: MR1L3:HOMS:ENV:RTD:2
        field: EGU C
        io: i
    '}
    fbMR1L3_Env_RTD_2 : FB_TempSensor;
    {attribute 'TcLinkTo' := '.iRaw := TIIB[MR1L3-EL3202-0010-E14]^RTD Inputs Channel 2^Value;
                              .bUnderrange := TIIB[MR1L3-EL3202-0010-E14]^RTD Inputs Channel 2^Status^Underrange;
                              .bOverrange := TIIB[MR1L3-EL3202-0010-E14]^RTD Inputs Channel 2^Status^Overrange;
                              .bError := TIIB[MR1L3-EL3202-0010-E14]^RTD Inputs Channel 2^Status^Error'}
    {attribute 'pytmc' := '
        pv: MR1L3:HOMS:ENV:RTD:3
        field: EGU C
        io: i
    '}
    fbMR1L3_Env_RTD_3 : FB_TempSensor;
    // MR2L3 RTDs
    {attribute 'TcLinkTo' := '.iRaw := TIIB[MR2L3-EL3202-0010-E13]^RTD Inputs Channel 1^Value;
                              .bUnderrange := TIIB[MR2L3-EL3202-0010-E13]^RTD Inputs Channel 1^Status^Underrange;
                              .bOverrange := TIIB[MR2L3-EL3202-0010-E13]^RTD Inputs Channel 1^Status^Overrange;
                              .bError := TIIB[MR2L3-EL3202-0010-E13]^RTD Inputs Channel 1^Status^Error'}
    {attribute 'pytmc' := '
        pv: MR2L3:HOMS:ENV:RTD:1
        field: EGU C
        io: i
    '}
    fbMR2L3_Env_RTD_1 : FB_TempSensor;
    {attribute 'TcLinkTo' := '.iRaw := TIIB[MR2L3-EL3202-0010-E14]^RTD Inputs Channel 1^Value;
                              .bUnderrange := TIIB[MR2L3-EL3202-0010-E14]^RTD Inputs Channel 1^Status^Underrange;
                              .bOverrange := TIIB[MR2L3-EL3202-0010-E14]^RTD Inputs Channel 1^Status^Overrange;
                              .bError := TIIB[MR2L3-EL3202-0010-E14]^RTD Inputs Channel 1^Status^Error'}
    {attribute 'pytmc' := '
        pv: MR2L3:HOMS:ENV:RTD:2
        field: EGU C
        io: i
    '}
    fbMR2L3_Env_RTD_2 : FB_TempSensor;
    {attribute 'TcLinkTo' := '.iRaw := TIIB[MR2L3-EL3202-0010-E14]^RTD Inputs Channel 2^Value;
                              .bUnderrange := TIIB[MR2L3-EL3202-0010-E14]^RTD Inputs Channel 2^Status^Underrange;
                              .bOverrange := TIIB[MR2L3-EL3202-0010-E14]^RTD Inputs Channel 2^Status^Overrange;
                              .bError := TIIB[MR2L3-EL3202-0010-E14]^RTD Inputs Channel 2^Status^Error'}
    {attribute 'pytmc' := '
        pv: MR2L3:HOMS:ENV:RTD:3
        field: EGU C
        io: i
    '}
    fbMR2L3_Env_RTD_3 : FB_TempSensor;
    // MR1L4 RTDs
    {attribute 'TcLinkTo' := '.iRaw := TIIB[MR1L4-EL3202-0010-E13]^RTD Inputs Channel 1^Value;
                              .bUnderrange := TIIB[MR1L4-EL3202-0010-E13]^RTD Inputs Channel 1^Status^Underrange;
                              .bOverrange := TIIB[MR1L4-EL3202-0010-E13]^RTD Inputs Channel 1^Status^Overrange;
                              .bError := TIIB[MR1L4-EL3202-0010-E13]^RTD Inputs Channel 1^Status^Error'}
    {attribute 'pytmc' := '
        pv: MR1L4:HOMS:ENV:RTD:1
        field: EGU C
        io: i
    '}
    fbMR1L4_Env_RTD_1 : FB_TempSensor;
    {attribute 'TcLinkTo' := '.iRaw := TIIB[MR1L4-EL3202-0010-E14]^RTD Inputs Channel 1^Value;
                              .bUnderrange := TIIB[MR1L4-EL3202-0010-E14]^RTD Inputs Channel 1^Status^Underrange;
                              .bOverrange := TIIB[MR1L4-EL3202-0010-E14]^RTD Inputs Channel 1^Status^Overrange;
                              .bError := TIIB[MR1L4-EL3202-0010-E14]^RTD Inputs Channel 1^Status^Error'}
    {attribute 'pytmc' := '
        pv: MR1L4:HOMS:ENV:RTD:2
        field: EGU C
        io: i
    '}
    fbMR1L4_Env_RTD_2 : FB_TempSensor;
    {attribute 'TcLinkTo' := '.iRaw := TIIB[MR1L4-EL3202-0010-E14]^RTD Inputs Channel 2^Value;
                              .bUnderrange := TIIB[MR1L4-EL3202-0010-E14]^RTD Inputs Channel 2^Status^Underrange;
                              .bOverrange := TIIB[MR1L4-EL3202-0010-E14]^RTD Inputs Channel 2^Status^Overrange;
                              .bError := TIIB[MR1L4-EL3202-0010-E14]^RTD Inputs Channel 2^Status^Error'}
    {attribute 'pytmc' := '
        pv: MR1L4:HOMS:ENV:RTD:3
        field: EGU C
        io: i
    '}
    fbMR1L4_Env_RTD_3 : FB_TempSensor;

END_VAR

// ---- GVLs/GVL_SerialIO.TcGVL
VAR_GLOBAL
    //Better have your inputs and outputs!
    //Serial_P1_stComIn   AT %I*	:	EL6inData22B (*KL6inData22B*);
    //Serial_P1_stComOut  AT %Q*	:	EL6outData22B (*KL6outData22B*);
     {attribute    'TcLinkTo'    :=    '.Status:=TIIB[EL6001_M1L3_PitchFine]^COM Inputs^Status;
                                 .D[0]:=TIIB[EL6001_M1L3_PitchFine]^COM Inputs^Data In 0;
                                 .D[1]:=TIIB[EL6001_M1L3_PitchFine]^COM Inputs^Data In 1;
                                 .D[2]:=TIIB[EL6001_M1L3_PitchFine]^COM Inputs^Data In 2;
                                 .D[3]:=TIIB[EL6001_M1L3_PitchFine]^COM Inputs^Data In 3;
                                 .D[4]:=TIIB[EL6001_M1L3_PitchFine]^COM Inputs^Data In 4;
                                 .D[5]:=TIIB[EL6001_M1L3_PitchFine]^COM Inputs^Data In 5;
                                 .D[6]:=TIIB[EL6001_M1L3_PitchFine]^COM Inputs^Data In 6;
                                 .D[7]:=TIIB[EL6001_M1L3_PitchFine]^COM Inputs^Data In 7;
                                 .D[8]:=TIIB[EL6001_M1L3_PitchFine]^COM Inputs^Data In 8;
                                 .D[9]:=TIIB[EL6001_M1L3_PitchFine]^COM Inputs^Data In 9;
                                 .D[10]:=TIIB[EL6001_M1L3_PitchFine]^COM Inputs^Data In 10;
                                 .D[11]:=TIIB[EL6001_M1L3_PitchFine]^COM Inputs^Data In 11;
                                 .D[12]:=TIIB[EL6001_M1L3_PitchFine]^COM Inputs^Data In 12;
                                 .D[13]:=TIIB[EL6001_M1L3_PitchFine]^COM Inputs^Data In 13;
                                 .D[14]:=TIIB[EL6001_M1L3_PitchFine]^COM Inputs^Data In 14;
                                 .D[15]:=TIIB[EL6001_M1L3_PitchFine]^COM Inputs^Data In 15;
                                 .D[16]:=TIIB[EL6001_M1L3_PitchFine]^COM Inputs^Data In 16;
                                 .D[17]:=TIIB[EL6001_M1L3_PitchFine]^COM Inputs^Data In 17;
                                 .D[18]:=TIIB[EL6001_M1L3_PitchFine]^COM Inputs^Data In 18;
                                 .D[19]:=TIIB[EL6001_M1L3_PitchFine]^COM Inputs^Data In 19;
                                 .D[20]:=TIIB[EL6001_M1L3_PitchFine]^COM Inputs^Data In 20;
                                 .D[21]:=TIIB[EL6001_M1L3_PitchFine]^COM Inputs^Data In 21;'}

Serial_stComIn_MR1L3 AT %I* : EL6inData22B; // M1L3 In Serial Comm Array
         {attribute    'TcLinkTo'    :=  '.D[0]:=TIIB[EL6001_M1L3_PitchFine]^COM Outputs^Data Out 0;
                                 .D[1]:=TIIB[EL6001_M1L3_PitchFine]^COM Outputs^Data Out 1;
                                 .D[2]:=TIIB[EL6001_M1L3_PitchFine]^COM Outputs^Data Out 2;
                                 .D[3]:=TIIB[EL6001_M1L3_PitchFine]^COM Outputs^Data Out 3;
                                 .D[4]:=TIIB[EL6001_M1L3_PitchFine]^COM Outputs^Data Out 4;
                                 .D[5]:=TIIB[EL6001_M1L3_PitchFine]^COM Outputs^Data Out 5;
                                 .D[6]:=TIIB[EL6001_M1L3_PitchFine]^COM Outputs^Data Out 6;
                                 .D[7]:=TIIB[EL6001_M1L3_PitchFine]^COM Outputs^Data Out 7;
                                 .D[8]:=TIIB[EL6001_M1L3_PitchFine]^COM Outputs^Data Out 8;
                                 .D[9]:=TIIB[EL6001_M1L3_PitchFine]^COM Outputs^Data Out 9;
                                 .D[10]:=TIIB[EL6001_M1L3_PitchFine]^COM Outputs^Data Out 10;
                                 .D[11]:=TIIB[EL6001_M1L3_PitchFine]^COM Outputs^Data Out 11;
                                 .D[12]:=TIIB[EL6001_M1L3_PitchFine]^COM Outputs^Data Out 12;
                                 .D[13]:=TIIB[EL6001_M1L3_PitchFine]^COM Outputs^Data Out 13;
                                 .D[14]:=TIIB[EL6001_M1L3_PitchFine]^COM Outputs^Data Out 14;
                                 .D[15]:=TIIB[EL6001_M1L3_PitchFine]^COM Outputs^Data Out 15;
                                 .D[16]:=TIIB[EL6001_M1L3_PitchFine]^COM Outputs^Data Out 16;
                                 .D[17]:=TIIB[EL6001_M1L3_PitchFine]^COM Outputs^Data Out 17;
                                 .D[18]:=TIIB[EL6001_M1L3_PitchFine]^COM Outputs^Data Out 18;
                                 .D[19]:=TIIB[EL6001_M1L3_PitchFine]^COM Outputs^Data Out 19;
                                 .D[20]:=TIIB[EL6001_M1L3_PitchFine]^COM Outputs^Data Out 20;
                                 .D[21]:=TIIB[EL6001_M1L3_PitchFine]^COM Outputs^Data Out 21;'}

    Serial_stComOut_MR1L3 AT %Q* : EL6outData22B; // M1 Out Serual Comm Array
         {attribute    'TcLinkTo'    :=    '.Status:=TIIB[EL6001_M1L4_PitchFine]^COM Inputs^Status;
                                 .D[0]:=TIIB[EL6001_M1L4_PitchFine]^COM Inputs^Data In 0;
                                 .D[1]:=TIIB[EL6001_M1L4_PitchFine]^COM Inputs^Data In 1;
                                 .D[2]:=TIIB[EL6001_M1L4_PitchFine]^COM Inputs^Data In 2;
                                 .D[3]:=TIIB[EL6001_M1L4_PitchFine]^COM Inputs^Data In 3;
                                 .D[4]:=TIIB[EL6001_M1L4_PitchFine]^COM Inputs^Data In 4;
                                 .D[5]:=TIIB[EL6001_M1L4_PitchFine]^COM Inputs^Data In 5;
                                 .D[6]:=TIIB[EL6001_M1L4_PitchFine]^COM Inputs^Data In 6;
                                 .D[7]:=TIIB[EL6001_M1L4_PitchFine]^COM Inputs^Data In 7;
                                 .D[8]:=TIIB[EL6001_M1L4_PitchFine]^COM Inputs^Data In 8;
                                 .D[9]:=TIIB[EL6001_M1L4_PitchFine]^COM Inputs^Data In 9;
                                 .D[10]:=TIIB[EL6001_M1L4_PitchFine]^COM Inputs^Data In 10;
                                 .D[11]:=TIIB[EL6001_M1L4_PitchFine]^COM Inputs^Data In 11;
                                 .D[12]:=TIIB[EL6001_M1L4_PitchFine]^COM Inputs^Data In 12;
                                 .D[13]:=TIIB[EL6001_M1L4_PitchFine]^COM Inputs^Data In 13;
                                 .D[14]:=TIIB[EL6001_M1L4_PitchFine]^COM Inputs^Data In 14;
                                 .D[15]:=TIIB[EL6001_M1L4_PitchFine]^COM Inputs^Data In 15;
                                 .D[16]:=TIIB[EL6001_M1L4_PitchFine]^COM Inputs^Data In 16;
                                 .D[17]:=TIIB[EL6001_M1L4_PitchFine]^COM Inputs^Data In 17;
                                 .D[18]:=TIIB[EL6001_M1L4_PitchFine]^COM Inputs^Data In 18;
                                 .D[19]:=TIIB[EL6001_M1L4_PitchFine]^COM Inputs^Data In 19;
                                 .D[20]:=TIIB[EL6001_M1L4_PitchFine]^COM Inputs^Data In 20;
                                 .D[21]:=TIIB[EL6001_M1L4_PitchFine]^COM Inputs^Data In 21;'}

